LIN {X 0,Y 354.923,Z 398.899,A -85,B 0,C 180,E1 -13512.581,E2 -13512.581} C_VEL
LIN {X 0,Y 354.894,Z 398.905,A -85,B 0,C 180,E1 -13516.096,E2 -13516.096} C_VEL
LIN {X 0,Y 354.908,Z 398.901,A -85,B 0,C 180,E1 -13518.472,E2 -13518.472} C_VEL
LIN {X 0,Y 354.836,Z 398.91,A -85,B 0,C 180,E1 -13522.106,E2 -13522.106} C_VEL
LIN {X 0,Y 354.9,Z 398.904,A -85,B 0,C 180,E1 -13525.827,E2 -13525.827} C_VEL
LIN {X 0,Y 354.819,Z 398.912,A -85,B 0,C 180,E1 -13529.682,E2 -13529.682} C_VEL
LIN {X 0,Y 354.807,Z 398.915,A -85,B 0,C 180,E1 -13533.702,E2 -13533.702} C_VEL
LIN {X 0,Y 354.803,Z 398.914,A -85,B 0,C 180,E1 -13536.459,E2 -13536.459} C_VEL
LIN {X 0,Y 354.825,Z 398.912,A -85,B 0,C 180,E1 -13539.424,E2 -13539.424} C_VEL
LIN {X 0,Y 354.79,Z 398.917,A -85,B 0,C 180,E1 -13542.867,E2 -13542.867} C_VEL
LIN {X 0,Y 354.779,Z 398.919,A -85,B 0,C 180,E1 -13546.105,E2 -13546.105} C_VEL
LIN {X 0,Y 354.854,Z 399.148,A -85,B 0,C 180,E1 -13547.122,E2 -13547.122} C_VEL
LIN {X 0,Y 355.19,Z 402.697,A -85,B 0,C 180,E1 -13550.505,E2 -13550.505} C_VEL
LIN {X 0,Y 355.149,Z 406.159,A -85,B 0,C 180,E1 -13553.582,E2 -13553.582} C_VEL
LIN {X 0,Y 354.934,Z 409.364,A -85,B 0,C 180,E1 -13556.329,E2 -13556.329} C_VEL
LIN {X 0,Y 354.662,Z 412.578,A -85,B 0,C 180,E1 -13558.988,E2 -13558.988} C_VEL
LIN {X 0,Y 354.41,Z 415.78,A -85,B 0,C 180,E1 -13561.581,E2 -13561.581} C_VEL
LIN {X 0,Y 354.107,Z 420.28,A -85,B 0,C 180,E1 -13565.134,E2 -13565.134} C_VEL
LIN {X 0,Y 358.979,Z 436.572,A -85,B 0,C 180,E1 -13566.069,E2 -13566.069} C_VEL
LIN {X 0,Y 362.051,Z 449.481,A -85,B 0,C 180,E1 -13566.956,E2 -13566.956} C_VEL
LIN {X 0,Y 363.817,Z 459.076,A -85,B 0,C 180,E1 -13567.713,E2 -13567.713} C_VEL
LIN {X 0,Y 363.535,Z 464.599,A -85,B 0,C 180,E1 -13568.119,E2 -13568.119} C_VEL
LIN {X 0,Y 362.37,Z 476.477,A -85,B 0,C 180,E1 -13569.122,E2 -13569.122} C_VEL
LIN {X 0,Y 360.894,Z 488.433,A -85,B 0,C 180,E1 -13570.371,E2 -13570.371} C_VEL
LIN {X 0,Y 359.361,Z 499.34,A -85,B 0,C 180,E1 -13571.765,E2 -13571.765} C_VEL
LIN {X 0,Y 357.822,Z 510.101,A -85,B 0,C 180,E1 -13573.453,E2 -13573.453} C_VEL
LIN {X 0,Y 356.582,Z 518.981,A -85,B 0,C 180,E1 -13575.154,E2 -13575.154} C_VEL
LIN {X 0,Y 355.662,Z 526.369,A -85,B 0,C 180,E1 -13576.865,E2 -13576.865} C_VEL
LIN {X 0,Y 354.749,Z 532.527,A -85,B 0,C 180,E1 -13578.574,E2 -13578.574} C_VEL
LIN {X 0,Y 354.17,Z 537.615,A -85,B 0,C 180,E1 -13580.29,E2 -13580.29} C_VEL
LIN {X 0,Y 353.634,Z 542.891,A -85,B 0,C 180,E1 -13582.578,E2 -13582.578} C_VEL
LIN {X 0,Y 353.426,Z 545.835,A -85,B 0,C 180,E1 -13584.294,E2 -13584.294} C_VEL
LIN {X 0,Y 353.232,Z 548.54,A -85,B 0,C 180,E1 -13586.578,E2 -13586.578} C_VEL
LIN {X 0,Y 353.157,Z 549.895,A -85,B 0,C 180,E1 -13588.86,E2 -13588.86} C_VEL
LIN {X 0,Y 353.157,Z 549.928,A -85,B 0,C 180,E1 -13591.14,E2 -13591.14} C_VEL
LIN {X 0,Y 353.231,Z 548.635,A -85,B 0,C 180,E1 -13593.422,E2 -13593.422} C_VEL
LIN {X 0,Y 353.424,Z 545.987,A -85,B 0,C 180,E1 -13595.706,E2 -13595.706} C_VEL
LIN {X 0,Y 353.721,Z 541.916,A -85,B 0,C 180,E1 -13597.995,E2 -13597.995} C_VEL
LIN {X 0,Y 354.314,Z 536.291,A -85,B 0,C 180,E1 -13600.284,E2 -13600.284} C_VEL
LIN {X 0,Y 355.115,Z 529.94,A -85,B 0,C 180,E1 -13602.284,E2 -13602.284} C_VEL
LIN {X 0,Y 356.245,Z 522.042,A -85,B 0,C 180,E1 -13604.277,E2 -13604.277} C_VEL
LIN {X 0,Y 357.339,Z 513.781,A -85,B 0,C 180,E1 -13605.983,E2 -13605.983} C_VEL
LIN {X 0,Y 358.781,Z 503.825,A -85,B 0,C 180,E1 -13607.675,E2 -13607.675} C_VEL
LIN {X 0,Y 360.336,Z 492.742,A -85,B 0,C 180,E1 -13609.216,E2 -13609.216} C_VEL
LIN {X 0,Y 361.75,Z 481.707,A -85,B 0,C 180,E1 -13610.469,E2 -13610.469} C_VEL
LIN {X 0,Y 363.134,Z 469.725,A -85,B 0,C 180,E1 -13611.575,E2 -13611.575} C_VEL
LIN {X 0,Y 363.949,Z 460.574,A -85,B 0,C 180,E1 -13612.269,E2 -13612.269} C_VEL
LIN {X 0,Y 362.131,Z 449.749,A -85,B 0,C 180,E1 -13613.128,E2 -13613.128} C_VEL
LIN {X 0,Y 358.864,Z 436.14,A -85,B 0,C 180,E1 -13614.063,E2 -13614.063} C_VEL
LIN {X 0,Y 354.669,Z 422.615,A -85,B 0,C 180,E1 -13614.849,E2 -13614.849} C_VEL
LIN {X 0,Y 354.099,Z 420.265,A -85,B 0,C 180,E1 -13614.985,E2 -13614.985} C_VEL
LIN {X 0,Y 354.31,Z 417.51,A -85,B 0,C 180,E1 -13617.144,E2 -13617.144} C_VEL
LIN {X 0,Y 354.66,Z 412.711,A -85,B 0,C 180,E1 -13621.012,E2 -13621.012} C_VEL
LIN {X 0,Y 354.928,Z 409.411,A -85,B 0,C 180,E1 -13623.731,E2 -13623.731} C_VEL
LIN {X 0,Y 355.142,Z 405.684,A -85,B 0,C 180,E1 -13626.92,E2 -13626.92} C_VEL
LIN {X 0,Y 354.513,Z 404.734,A -85,B 0,C 180,E1 -13627.855,E2 -13627.855} C_VEL
LIN {X 0,Y 351.722,Z 403.491,A -85,B 0,C 180,E1 -13629.385,E2 -13629.385} C_VEL
LIN {X 0,Y 349.277,Z 402.535,A -85,B 0,C 180,E1 -13630.623,E2 -13630.623} C_VEL
LIN {X 0,Y 348.133,Z 401.704,A -85,B 0,C 180,E1 -13631.578,E2 -13631.578} C_VEL
LIN {X 0,Y 347.99,Z 401.39,A -85,B 0,C 180,E1 -13631.901,E2 -13631.901} C_VEL
LIN {X 0,Y 347.786,Z 399.889,A -85,B 0,C 180,E1 -13633.399,E2 -13633.399} C_VEL
LIN {X 0,Y 347.728,Z 399.801,A -85,B 0,C 180,E1 -13636.686,E2 -13636.686} C_VEL
LIN {X 0,Y 347.749,Z 399.794,A -85,B 0,C 180,E1 -13640.173,E2 -13640.173} C_VEL
LIN {X 0,Y 347.765,Z 399.793,A -85,B 0,C 180,E1 -13642.679,E2 -13642.679} C_VEL
LIN {X 0,Y 347.75,Z 399.793,A -85,B 0,C 180,E1 -13645.956,E2 -13645.956} C_VEL
LIN {X 0,Y 347.766,Z 399.791,A -85,B 0,C 180,E1 -13649.654,E2 -13649.654} C_VEL
LIN {X 0,Y 347.853,Z 399.782,A -85,B 0,C 180,E1 -13652.745,E2 -13652.745} C_VEL
LIN {X 0,Y 347.791,Z 399.785,A -85,B 0,C 180,E1 -13656.162,E2 -13656.162} C_VEL
LIN {X 0,Y 347.82,Z 399.779,A -85,B 0,C 180,E1 -13659.91,E2 -13659.91} C_VEL
LIN {X 0,Y 347.869,Z 399.779,A -85,B 0,C 180,E1 -13662.359,E2 -13662.359} C_VEL
LIN {X 0,Y 347.9,Z 399.773,A -85,B 0,C 180,E1 -13665.971,E2 -13665.971} C_VEL
LIN {X 0,Y 347.931,Z 399.769,A -85,B 0,C 180,E1 -13669.526,E2 -13669.526} C_VEL
LIN {X 0,Y 348.077,Z 399.753,A -85,B 0,C 180,E1 -13671.875,E2 -13671.875} C_VEL
LIN {X 0,Y 348.07,Z 399.752,A -85,B 0,C 180,E1 -13674.206,E2 -13674.206} C_VEL
LIN {X 0,Y 348.209,Z 399.735,A -85,B 0,C 180,E1 -13677.686,E2 -13677.686} C_VEL
LIN {X 0,Y 348.348,Z 399.721,A -85,B 0,C 180,E1 -13680,E2 -13680} C_VEL
LIN {X 0,Y 348.211,Z 399.735,A -85,B 0,C 180,E1 -13682.313,E2 -13682.313} C_VEL
LIN {X 0,Y 348.109,Z 399.748,A -85,B 0,C 180,E1 -13686.957,E2 -13686.957} C_VEL
LIN {X 0,Y 347.971,Z 399.766,A -85,B 0,C 180,E1 -13689.298,E2 -13689.298} C_VEL
LIN {X 0,Y 347.893,Z 399.776,A -85,B 0,C 180,E1 -13692.839,E2 -13692.839} C_VEL
LIN {X 0,Y 347.842,Z 399.782,A -85,B 0,C 180,E1 -13696.431,E2 -13696.431} C_VEL
LIN {X 0,Y 347.858,Z 399.779,A -85,B 0,C 180,E1 -13698.86,E2 -13698.86} C_VEL
LIN {X 0,Y 347.776,Z 399.791,A -85,B 0,C 180,E1 -13702.579,E2 -13702.579} C_VEL
LIN {X 0,Y 347.814,Z 399.784,A -85,B 0,C 180,E1 -13705.108,E2 -13705.108} C_VEL
LIN {X 0,Y 347.81,Z 399.784,A -85,B 0,C 180,E1 -13707.694,E2 -13707.694} C_VEL
LIN {X 0,Y 347.751,Z 399.79,A -85,B 0,C 180,E1 -13710.348,E2 -13710.348} C_VEL
LIN {X 0,Y 347.75,Z 399.796,A -85,B 0,C 180,E1 -13714.044,E2 -13714.044} C_VEL
LIN {X 0,Y 347.769,Z 399.796,A -85,B 0,C 180,E1 -13717.32,E2 -13717.32} C_VEL
LIN {X 0,Y 347.757,Z 399.797,A -85,B 0,C 180,E1 -13720.294,E2 -13720.294} C_VEL
LIN {X 0,Y 347.785,Z 399.804,A -85,B 0,C 180,E1 -13723.999,E2 -13723.999} C_VEL
LIN {X 0,Y 348.233,Z 402.702,A -85,B 0,C 180,E1 -13726.671,E2 -13726.671} C_VEL
LIN {X 0,Y 348.67,Z 406.35,A -85,B 0,C 180,E1 -13729.833,E2 -13729.833} C_VEL
LIN {X 0,Y 348.579,Z 409.986,A -85,B 0,C 180,E1 -13732.781,E2 -13732.781} C_VEL
LIN {X 0,Y 348.24,Z 413.96,A -85,B 0,C 180,E1 -13735.837,E2 -13735.837} C_VEL
LIN {X 0,Y 347.717,Z 419.139,A -85,B 0,C 180,E1 -13739.649,E2 -13739.649} C_VEL
LIN {X 0,Y 347.25,Z 424.619,A -85,B 0,C 180,E1 -13743.56,E2 -13743.56} C_VEL
LIN {X 0,Y 347.141,Z 426.014,A -85,B 0,C 180,E1 -13744.533,E2 -13744.533} C_VEL
LIN {X 0,Y 351.781,Z 442.131,A -85,B 0,C 180,E1 -13745.454,E2 -13745.454} C_VEL
LIN {X 0,Y 354.766,Z 455.294,A -85,B 0,C 180,E1 -13746.359,E2 -13746.359} C_VEL
LIN {X 0,Y 356.927,Z 468.457,A -85,B 0,C 180,E1 -13747.423,E2 -13747.423} C_VEL
LIN {X 0,Y 355.707,Z 481.093,A -85,B 0,C 180,E1 -13748.465,E2 -13748.465} C_VEL
LIN {X 0,Y 354.168,Z 492.999,A -85,B 0,C 180,E1 -13749.68,E2 -13749.68} C_VEL
LIN {X 0,Y 352.564,Z 504.301,A -85,B 0,C 180,E1 -13751.099,E2 -13751.099} C_VEL
LIN {X 0,Y 350.942,Z 515.371,A -85,B 0,C 180,E1 -13752.819,E2 -13752.819} C_VEL
LIN {X 0,Y 349.61,Z 524.504,A -85,B 0,C 180,E1 -13754.552,E2 -13754.552} C_VEL
LIN {X 0,Y 348.47,Z 533.233,A -85,B 0,C 180,E1 -13756.589,E2 -13756.589} C_VEL
LIN {X 0,Y 347.515,Z 539.378,A -85,B 0,C 180,E1 -13758.332,E2 -13758.332} C_VEL
LIN {X 0,Y 346.806,Z 545.907,A -85,B 0,C 180,E1 -13760.67,E2 -13760.67} C_VEL
LIN {X 0,Y 346.342,Z 550.793,A -85,B 0,C 180,E1 -13763.007,E2 -13763.007} C_VEL
LIN {X 0,Y 346.157,Z 554.19,A -85,B 0,C 180,E1 -13765.342,E2 -13765.342} C_VEL
LIN {X 0,Y 346.045,Z 556.198,A -85,B 0,C 180,E1 -13767.672,E2 -13767.672} C_VEL
LIN {X 0,Y 346.074,Z 556.862,A -85,B 0,C 180,E1 -13770,E2 -13770} C_VEL
LIN {X 0,Y 346.045,Z 556.192,A -85,B 0,C 180,E1 -13772.328,E2 -13772.328} C_VEL
LIN {X 0,Y 346.16,Z 554.18,A -85,B 0,C 180,E1 -13774.658,E2 -13774.658} C_VEL
LIN {X 0,Y 346.371,Z 550.776,A -85,B 0,C 180,E1 -13776.993,E2 -13776.993} C_VEL
LIN {X 0,Y 346.786,Z 545.877,A -85,B 0,C 180,E1 -13779.33,E2 -13779.33} C_VEL
LIN {X 0,Y 347.315,Z 541.154,A -85,B 0,C 180,E1 -13781.083,E2 -13781.083} C_VEL
LIN {X 0,Y 348.309,Z 534.306,A -85,B 0,C 180,E1 -13783.12,E2 -13783.12} C_VEL
LIN {X 0,Y 349.38,Z 525.802,A -85,B 0,C 180,E1 -13785.159,E2 -13785.159} C_VEL
LIN {X 0,Y 350.687,Z 516.931,A -85,B 0,C 180,E1 -13786.893,E2 -13786.893} C_VEL
LIN {X 0,Y 352.278,Z 506.184,A -85,B 0,C 180,E1 -13788.615,E2 -13788.615} C_VEL
LIN {X 0,Y 353.858,Z 495.308,A -85,B 0,C 180,E1 -13790.036,E2 -13790.036} C_VEL
LIN {X 0,Y 355.434,Z 483.058,A -85,B 0,C 180,E1 -13791.341,E2 -13791.341} C_VEL
LIN {X 0,Y 356.807,Z 470.278,A -85,B 0,C 180,E1 -13792.429,E2 -13792.429} C_VEL
LIN {X 0,Y 356.602,Z 466.361,A -85,B 0,C 180,E1 -13792.745,E2 -13792.745} C_VEL
LIN {X 0,Y 354.228,Z 452.721,A -85,B 0,C 180,E1 -13793.816,E2 -13793.816} C_VEL
LIN {X 0,Y 351.015,Z 439.421,A -85,B 0,C 180,E1 -13794.703,E2 -13794.703} C_VEL
LIN {X 0,Y 347.23,Z 426.891,A -85,B 0,C 180,E1 -13795.406,E2 -13795.406} C_VEL
LIN {X 0,Y 347.125,Z 426.008,A -85,B 0,C 180,E1 -13795.456,E2 -13795.456} C_VEL
LIN {X 0,Y 347.564,Z 420.929,A -85,B 0,C 180,E1 -13799.032,E2 -13799.032} C_VEL
LIN {X 0,Y 348.081,Z 415.449,A -85,B 0,C 180,E1 -13803.035,E2 -13803.035} C_VEL
LIN {X 0,Y 348.502,Z 411.233,A -85,B 0,C 180,E1 -13806.23,E2 -13806.23} C_VEL
LIN {X 0,Y 348.675,Z 408.132,A -85,B 0,C 180,E1 -13808.671,E2 -13808.671} C_VEL
LIN {X 0,Y 348.668,Z 406.318,A -85,B 0,C 180,E1 -13810.167,E2 -13810.167} C_VEL
LIN {X 0,Y 348.201,Z 402.67,A -85,B 0,C 180,E1 -13813.334,E2 -13813.334} C_VEL
LIN {X 0,Y 347.784,Z 399.794,A -85,B 0,C 180,E1 -13816.001,E2 -13816.001} C_VEL
LIN {X 0,Y 347.756,Z 399.795,A -85,B 0,C 180,E1 -13819.706,E2 -13819.706} C_VEL
LIN {X 0,Y 347.768,Z 399.794,A -85,B 0,C 180,E1 -13822.68,E2 -13822.68} C_VEL
LIN {X 0,Y 347.749,Z 399.796,A -85,B 0,C 180,E1 -13825.956,E2 -13825.956} C_VEL
LIN {X 0,Y 347.75,Z 399.795,A -85,B 0,C 180,E1 -13829.652,E2 -13829.652} C_VEL
LIN {X 0,Y 347.831,Z 399.784,A -85,B 0,C 180,E1 -13833.608,E2 -13833.608} C_VEL
LIN {X 0,Y 347.786,Z 399.789,A -85,B 0,C 180,E1 -13836.162,E2 -13836.162} C_VEL
LIN {X 0,Y 347.813,Z 399.784,A -85,B 0,C 180,E1 -13839.909,E2 -13839.909} C_VEL
LIN {X 0,Y 347.868,Z 399.777,A -85,B 0,C 180,E1 -13842.359,E2 -13842.359} C_VEL
LIN {X 0,Y 347.898,Z 399.773,A -85,B 0,C 180,E1 -13845.971,E2 -13845.971} C_VEL
LIN {X 0,Y 347.93,Z 399.767,A -85,B 0,C 180,E1 -13849.526,E2 -13849.526} C_VEL
LIN {X 0,Y 348.076,Z 399.751,A -85,B 0,C 180,E1 -13851.875,E2 -13851.875} C_VEL
LIN {X 0,Y 348.069,Z 399.752,A -85,B 0,C 180,E1 -13854.206,E2 -13854.206} C_VEL
LIN {X 0,Y 348.21,Z 399.734,A -85,B 0,C 180,E1 -13857.687,E2 -13857.687} C_VEL
LIN {X 0,Y 348.369,Z 399.717,A -85,B 0,C 180,E1 -13860,E2 -13860} C_VEL
LIN {X 0,Y 348.208,Z 399.734,A -85,B 0,C 180,E1 -13862.314,E2 -13862.314} C_VEL
LIN {X 0,Y 348.108,Z 399.748,A -85,B 0,C 180,E1 -13866.958,E2 -13866.958} C_VEL
LIN {X 0,Y 347.97,Z 399.765,A -85,B 0,C 180,E1 -13869.299,E2 -13869.299} C_VEL
LIN {X 0,Y 347.892,Z 399.774,A -85,B 0,C 180,E1 -13872.84,E2 -13872.84} C_VEL
LIN {X 0,Y 347.843,Z 399.779,A -85,B 0,C 180,E1 -13876.431,E2 -13876.431} C_VEL
LIN {X 0,Y 347.857,Z 399.779,A -85,B 0,C 180,E1 -13878.86,E2 -13878.86} C_VEL
LIN {X 0,Y 347.776,Z 399.792,A -85,B 0,C 180,E1 -13882.579,E2 -13882.579} C_VEL
LIN {X 0,Y 347.813,Z 399.784,A -85,B 0,C 180,E1 -13885.108,E2 -13885.108} C_VEL
LIN {X 0,Y 347.809,Z 399.788,A -85,B 0,C 180,E1 -13887.694,E2 -13887.694} C_VEL
LIN {X 0,Y 347.75,Z 399.792,A -85,B 0,C 180,E1 -13890.348,E2 -13890.348} C_VEL
LIN {X 0,Y 347.749,Z 399.795,A -85,B 0,C 180,E1 -13894.044,E2 -13894.044} C_VEL
LIN {X 0,Y 347.767,Z 399.793,A -85,B 0,C 180,E1 -13897.32,E2 -13897.32} C_VEL
LIN {X 0,Y 347.734,Z 399.796,A -85,B 0,C 180,E1 -13900.297,E2 -13900.297} C_VEL
LIN {X 0,Y 347.727,Z 399.797,A -85,B 0,C 180,E1 -13903.408,E2 -13903.408} C_VEL
LIN {X 0,Y 347.778,Z 399.85,A -85,B 0,C 180,E1 -13906.677,E2 -13906.677} C_VEL
LIN {X 0,Y 348.152,Z 403.345,A -85,B 0,C 180,E1 -13910.094,E2 -13910.094} C_VEL
LIN {X 0,Y 348.127,Z 406.196,A -85,B 0,C 180,E1 -13912.725,E2 -13912.725} C_VEL
LIN {X 0,Y 347.921,Z 409.844,A -85,B 0,C 180,E1 -13915.915,E2 -13915.915} C_VEL
LIN {X 0,Y 347.545,Z 414.23,A -85,B 0,C 180,E1 -13919.632,E2 -13919.632} C_VEL
LIN {X 0,Y 347.205,Z 419.05,A -85,B 0,C 180,E1 -13923.557,E2 -13923.557} C_VEL
LIN {X 0,Y 347.099,Z 420.355,A -85,B 0,C 180,E1 -13924.602,E2 -13924.602} C_VEL
LIN {X 0,Y 352.04,Z 436.533,A -85,B 0,C 180,E1 -13925.561,E2 -13925.561} C_VEL
LIN {X 0,Y 355.127,Z 449.404,A -85,B 0,C 180,E1 -13926.47,E2 -13926.47} C_VEL
LIN {X 0,Y 357.249,Z 461.563,A -85,B 0,C 180,E1 -13927.466,E2 -13927.466} C_VEL
LIN {X 0,Y 355.922,Z 475.051,A -85,B 0,C 180,E1 -13928.574,E2 -13928.574} C_VEL
LIN {X 0,Y 354.375,Z 487.327,A -85,B 0,C 180,E1 -13929.844,E2 -13929.844} C_VEL
LIN {X 0,Y 352.844,Z 497.419,A -85,B 0,C 180,E1 -13931.115,E2 -13931.115} C_VEL
LIN {X 0,Y 351.507,Z 506.838,A -85,B 0,C 180,E1 -13932.548,E2 -13932.548} C_VEL
LIN {X 0,Y 350.09,Z 516.305,A -85,B 0,C 180,E1 -13934.276,E2 -13934.276} C_VEL
LIN {X 0,Y 348.91,Z 525.327,A -85,B 0,C 180,E1 -13936.31,E2 -13936.31} C_VEL
LIN {X 0,Y 347.752,Z 532.598,A -85,B 0,C 180,E1 -13938.34,E2 -13938.34} C_VEL
LIN {X 0,Y 347.135,Z 537.686,A -85,B 0,C 180,E1 -13940.091,E2 -13940.091} C_VEL
LIN {X 0,Y 346.56,Z 542.961,A -85,B 0,C 180,E1 -13942.426,E2 -13942.426} C_VEL
LIN {X 0,Y 346.345,Z 545.904,A -85,B 0,C 180,E1 -13944.177,E2 -13944.177} C_VEL
LIN {X 0,Y 346.159,Z 548.609,A -85,B 0,C 180,E1 -13946.508,E2 -13946.508} C_VEL
LIN {X 0,Y 346.06,Z 549.964,A -85,B 0,C 180,E1 -13948.836,E2 -13948.836} C_VEL
LIN {X 0,Y 346.06,Z 549.997,A -85,B 0,C 180,E1 -13951.164,E2 -13951.164} C_VEL
LIN {X 0,Y 346.158,Z 548.704,A -85,B 0,C 180,E1 -13953.492,E2 -13953.492} C_VEL
LIN {X 0,Y 346.341,Z 546.055,A -85,B 0,C 180,E1 -13955.823,E2 -13955.823} C_VEL
LIN {X 0,Y 346.663,Z 541.984,A -85,B 0,C 180,E1 -13958.159,E2 -13958.159} C_VEL
LIN {X 0,Y 347.303,Z 536.359,A -85,B 0,C 180,E1 -13960.494,E2 -13960.494} C_VEL
LIN {X 0,Y 348.178,Z 530.007,A -85,B 0,C 180,E1 -13962.532,E2 -13962.532} C_VEL
LIN {X 0,Y 349.2,Z 523.337,A -85,B 0,C 180,E1 -13964.273,E2 -13964.273} C_VEL
LIN {X 0,Y 350.255,Z 515.478,A -85,B 0,C 180,E1 -13965.986,E2 -13965.986} C_VEL
LIN {X 0,Y 351.728,Z 505.67,A -85,B 0,C 180,E1 -13967.741,E2 -13967.741} C_VEL
LIN {X 0,Y 353.314,Z 494.948,A -85,B 0,C 180,E1 -13969.311,E2 -13969.311} C_VEL
LIN {X 0,Y 354.92,Z 483.066,A -85,B 0,C 180,E1 -13970.73,E2 -13970.73} C_VEL
LIN {X 0,Y 356.347,Z 471.396,A -85,B 0,C 180,E1 -13971.854,E2 -13971.854} C_VEL
LIN {X 0,Y 357.243,Z 460.637,A -85,B 0,C 180,E1 -13972.711,E2 -13972.711} C_VEL
LIN {X 0,Y 354.86,Z 448.199,A -85,B 0,C 180,E1 -13973.726,E2 -13973.726} C_VEL
LIN {X 0,Y 351.56,Z 434.852,A -85,B 0,C 180,E1 -13974.654,E2 -13974.654} C_VEL
LIN {X 0,Y 347.095,Z 420.357,A -85,B 0,C 180,E1 -13975.505,E2 -13975.505} C_VEL
LIN {X 0,Y 347.407,Z 415.979,A -85,B 0,C 180,E1 -13979.047,E2 -13979.047} C_VEL
LIN {X 0,Y 347.695,Z 412.513,A -85,B 0,C 180,E1 -13981.902,E2 -13981.902} C_VEL
LIN {X 0,Y 347.925,Z 409.517,A -85,B 0,C 180,E1 -13984.444,E2 -13984.444} C_VEL
LIN {X 0,Y 348.129,Z 406.326,A -85,B 0,C 180,E1 -13987.275,E2 -13987.275} C_VEL
LIN {X 0,Y 348.144,Z 403.115,A -85,B 0,C 180,E1 -13990.24,E2 -13990.24} C_VEL
LIN {X 0,Y 347.99,Z 401.39,A -85,B 0,C 180,E1 -13991.901,E2 -13991.901} C_VEL
LIN {X 0,Y 347.159,Z 400.689,A -85,B 0,C 180,E1 -13992.857,E2 -13992.857} C_VEL
LIN {X 0,Y 344.17,Z 400.394,A -85,B 0,C 180,E1 -13994.423,E2 -13994.423} C_VEL
LIN {X 0,Y 341.743,Z 400.551,A -85,B 0,C 180,E1 -13995.697,E2 -13995.697} C_VEL
LIN {X 0,Y 340.74,Z 400.672,A -85,B 0,C 180,E1 -13996.683,E2 -13996.683} C_VEL
LIN {X 0,Y 340.674,Z 400.679,A -85,B 0,C 180,E1 -13997.017,E2 -13997.017} C_VEL
LIN {X 0,Y 340.701,Z 400.672,A -85,B 0,C 180,E1 -14000.248,E2 -14000.248} C_VEL
LIN {X 0,Y 340.713,Z 400.669,A -85,B 0,C 180,E1 -14003.559,E2 -14003.559} C_VEL
LIN {X 0,Y 340.696,Z 400.673,A -85,B 0,C 180,E1 -14006.154,E2 -14006.154} C_VEL
LIN {X 0,Y 340.777,Z 400.661,A -85,B 0,C 180,E1 -14010.333,E2 -14010.333} C_VEL
LIN {X 0,Y 340.806,Z 400.658,A -85,B 0,C 180,E1 -14013.02,E2 -14013.02} C_VEL
LIN {X 0,Y 340.731,Z 400.665,A -85,B 0,C 180,E1 -14016.927,E2 -14016.927} C_VEL
LIN {X 0,Y 340.797,Z 400.66,A -85,B 0,C 180,E1 -14020.734,E2 -14020.734} C_VEL
LIN {X 0,Y 340.789,Z 400.659,A -85,B 0,C 180,E1 -14023.219,E2 -14023.219} C_VEL
LIN {X 0,Y 340.847,Z 400.653,A -85,B 0,C 180,E1 -14026.89,E2 -14026.89} C_VEL
LIN {X 0,Y 340.931,Z 400.642,A -85,B 0,C 180,E1 -14030.508,E2 -14030.508} C_VEL
LIN {X 0,Y 341.079,Z 400.623,A -85,B 0,C 180,E1 -14032.898,E2 -14032.898} C_VEL
LIN {X 0,Y 341.171,Z 400.612,A -85,B 0,C 180,E1 -14037.639,E2 -14037.639} C_VEL
LIN {X 0,Y 341.298,Z 400.599,A -85,B 0,C 180,E1 -14040,E2 -14040} C_VEL
LIN {X 0,Y 341.173,Z 400.612,A -85,B 0,C 180,E1 -14042.361,E2 -14042.361} C_VEL
LIN {X 0,Y 341.079,Z 400.623,A -85,B 0,C 180,E1 -14047.102,E2 -14047.102} C_VEL
LIN {X 0,Y 340.875,Z 400.648,A -85,B 0,C 180,E1 -14050.694,E2 -14050.694} C_VEL
LIN {X 0,Y 340.865,Z 400.652,A -85,B 0,C 180,E1 -14054.325,E2 -14054.325} C_VEL
LIN {X 0,Y 340.84,Z 400.653,A -85,B 0,C 180,E1 -14058.467,E2 -14058.467} C_VEL
LIN {X 0,Y 340.756,Z 400.664,A -85,B 0,C 180,E1 -14061.857,E2 -14061.857} C_VEL
LIN {X 0,Y 340.774,Z 400.662,A -85,B 0,C 180,E1 -14065.664,E2 -14065.664} C_VEL
LIN {X 0,Y 340.73,Z 400.667,A -85,B 0,C 180,E1 -14068.321,E2 -14068.321} C_VEL
LIN {X 0,Y 340.7,Z 400.673,A -85,B 0,C 180,E1 -14071.044,E2 -14071.044} C_VEL
LIN {X 0,Y 340.721,Z 400.671,A -85,B 0,C 180,E1 -14075.279,E2 -14075.279} C_VEL
LIN {X 0,Y 340.722,Z 400.673,A -85,B 0,C 180,E1 -14078.388,E2 -14078.388} C_VEL
LIN {X 0,Y 340.735,Z 400.671,A -85,B 0,C 180,E1 -14082.052,E2 -14082.052} C_VEL
LIN {X 0,Y 340.757,Z 400.84,A -85,B 0,C 180,E1 -14083.791,E2 -14083.791} C_VEL
LIN {X 0,Y 341.295,Z 404.475,A -85,B 0,C 180,E1 -14087.192,E2 -14087.192} C_VEL
LIN {X 0,Y 341.657,Z 408.115,A -85,B 0,C 180,E1 -14090.381,E2 -14090.381} C_VEL
LIN {X 0,Y 341.514,Z 411.77,A -85,B 0,C 180,E1 -14093.377,E2 -14093.377} C_VEL
LIN {X 0,Y 341.131,Z 415.42,A -85,B 0,C 180,E1 -14096.202,E2 -14096.202} C_VEL
LIN {X 0,Y 340.615,Z 420.564,A -85,B 0,C 180,E1 -14100.066,E2 -14100.066} C_VEL
LIN {X 0,Y 340.134,Z 425.958,A -85,B 0,C 180,E1 -14103.983,E2 -14103.983} C_VEL
LIN {X 0,Y 341.878,Z 431.912,A -85,B 0,C 180,E1 -14104.295,E2 -14104.295} C_VEL
LIN {X 0,Y 345.815,Z 445.867,A -85,B 0,C 180,E1 -14105.18,E2 -14105.18} C_VEL
LIN {X 0,Y 348.571,Z 458.794,A -85,B 0,C 180,E1 -14106.14,E2 -14106.14} C_VEL
LIN {X 0,Y 350.244,Z 470.619,A -85,B 0,C 180,E1 -14107.147,E2 -14107.147} C_VEL
LIN {X 0,Y 348.795,Z 483.48,A -85,B 0,C 180,E1 -14108.271,E2 -14108.271} C_VEL
LIN {X 0,Y 347.136,Z 495.346,A -85,B 0,C 180,E1 -14109.559,E2 -14109.559} C_VEL
LIN {X 0,Y 345.518,Z 506.203,A -85,B 0,C 180,E1 -14111.007,E2 -14111.007} C_VEL
LIN {X 0,Y 343.862,Z 516.933,A -85,B 0,C 180,E1 -14112.761,E2 -14112.761} C_VEL
LIN {X 0,Y 342.511,Z 525.792,A -85,B 0,C 180,E1 -14114.529,E2 -14114.529} C_VEL
LIN {X 0,Y 341.517,Z 533.165,A -85,B 0,C 180,E1 -14116.311,E2 -14116.311} C_VEL
LIN {X 0,Y 340.537,Z 539.31,A -85,B 0,C 180,E1 -14118.09,E2 -14118.09} C_VEL
LIN {X 0,Y 339.764,Z 545.839,A -85,B 0,C 180,E1 -14120.475,E2 -14120.475} C_VEL
LIN {X 0,Y 339.272,Z 550.725,A -85,B 0,C 180,E1 -14122.86,E2 -14122.86} C_VEL
LIN {X 0,Y 339.064,Z 554.121,A -85,B 0,C 180,E1 -14125.244,E2 -14125.244} C_VEL
LIN {X 0,Y 338.961,Z 556.129,A -85,B 0,C 180,E1 -14127.623,E2 -14127.623} C_VEL
LIN {X 0,Y 338.977,Z 556.793,A -85,B 0,C 180,E1 -14130,E2 -14130} C_VEL
LIN {X 0,Y 338.961,Z 556.123,A -85,B 0,C 180,E1 -14132.377,E2 -14132.377} C_VEL
LIN {X 0,Y 339.066,Z 554.11,A -85,B 0,C 180,E1 -14134.756,E2 -14134.756} C_VEL
LIN {X 0,Y 339.29,Z 550.706,A -85,B 0,C 180,E1 -14137.139,E2 -14137.139} C_VEL
LIN {X 0,Y 339.749,Z 545.807,A -85,B 0,C 180,E1 -14139.525,E2 -14139.525} C_VEL
LIN {X 0,Y 340.535,Z 539.27,A -85,B 0,C 180,E1 -14141.91,E2 -14141.91} C_VEL
LIN {X 0,Y 341.625,Z 531.998,A -85,B 0,C 180,E1 -14143.988,E2 -14143.988} C_VEL
LIN {X 0,Y 342.945,Z 522.989,A -85,B 0,C 180,E1 -14146.061,E2 -14146.061} C_VEL
LIN {X 0,Y 344.417,Z 513.536,A -85,B 0,C 180,E1 -14147.823,E2 -14147.823} C_VEL
LIN {X 0,Y 346.016,Z 503.07,A -85,B 0,C 180,E1 -14149.426,E2 -14149.426} C_VEL
LIN {X 0,Y 347.704,Z 491.52,A -85,B 0,C 180,E1 -14150.87,E2 -14150.87} C_VEL
LIN {X 0,Y 349.273,Z 478.889,A -85,B 0,C 180,E1 -14152.147,E2 -14152.147} C_VEL
LIN {X 0,Y 350.172,Z 470.5,A -85,B 0,C 180,E1 -14152.853,E2 -14152.853} C_VEL
LIN {X 0,Y 348.423,Z 458.217,A -85,B 0,C 180,E1 -14153.894,E2 -14153.894} C_VEL
LIN {X 0,Y 345.412,Z 444.356,A -85,B 0,C 180,E1 -14154.911,E2 -14154.911} C_VEL
LIN {X 0,Y 341.509,Z 430.874,A -85,B 0,C 180,E1 -14155.752,E2 -14155.752} C_VEL
LIN {X 0,Y 340.117,Z 425.934,A -85,B 0,C 180,E1 -14156.018,E2 -14156.018} C_VEL
LIN {X 0,Y 340.596,Z 420.876,A -85,B 0,C 180,E1 -14159.685,E2 -14159.685} C_VEL
LIN {X 0,Y 340.944,Z 417.206,A -85,B 0,C 180,E1 -14162.408,E2 -14162.408} C_VEL
LIN {X 0,Y 341.315,Z 413.555,A -85,B 0,C 180,E1 -14165.208,E2 -14165.208} C_VEL
LIN {X 0,Y 341.601,Z 409.906,A -85,B 0,C 180,E1 -14168.113,E2 -14168.113} C_VEL
LIN {X 0,Y 341.613,Z 407.142,A -85,B 0,C 180,E1 -14170.43,E2 -14170.43} C_VEL
LIN {X 0,Y 341.129,Z 403.297,A -85,B 0,C 180,E1 -14173.857,E2 -14173.857} C_VEL
LIN {X 0,Y 340.741,Z 400.671,A -85,B 0,C 180,E1 -14176.434,E2 -14176.434} C_VEL
LIN {X 0,Y 340.711,Z 400.672,A -85,B 0,C 180,E1 -14180.249,E2 -14180.249} C_VEL
LIN {X 0,Y 340.713,Z 400.671,A -85,B 0,C 180,E1 -14183.559,E2 -14183.559} C_VEL
LIN {X 0,Y 340.695,Z 400.675,A -85,B 0,C 180,E1 -14186.154,E2 -14186.154} C_VEL
LIN {X 0,Y 340.742,Z 400.668,A -85,B 0,C 180,E1 -14190.329,E2 -14190.329} C_VEL
LIN {X 0,Y 340.804,Z 400.659,A -85,B 0,C 180,E1 -14193.02,E2 -14193.02} C_VEL
LIN {X 0,Y 340.755,Z 400.666,A -85,B 0,C 180,E1 -14195.638,E2 -14195.638} C_VEL
LIN {X 0,Y 340.738,Z 400.666,A -85,B 0,C 180,E1 -14199.474,E2 -14199.474} C_VEL
LIN {X 0,Y 340.86,Z 400.65,A -85,B 0,C 180,E1 -14201.984,E2 -14201.984} C_VEL
LIN {X 0,Y 340.87,Z 400.648,A -85,B 0,C 180,E1 -14205.705,E2 -14205.705} C_VEL
LIN {X 0,Y 340.872,Z 400.646,A -85,B 0,C 180,E1 -14209.306,E2 -14209.306} C_VEL
LIN {X 0,Y 341.077,Z 400.619,A -85,B 0,C 180,E1 -14212.898,E2 -14212.898} C_VEL
LIN {X 0,Y 341.172,Z 400.611,A -85,B 0,C 180,E1 -14217.639,E2 -14217.639} C_VEL
LIN {X 0,Y 341.318,Z 400.595,A -85,B 0,C 180,E1 -14220,E2 -14220} C_VEL
LIN {X 0,Y 341.169,Z 400.611,A -85,B 0,C 180,E1 -14222.361,E2 -14222.361} C_VEL
LIN {X 0,Y 341.077,Z 400.624,A -85,B 0,C 180,E1 -14227.102,E2 -14227.102} C_VEL
LIN {X 0,Y 340.874,Z 400.648,A -85,B 0,C 180,E1 -14230.694,E2 -14230.694} C_VEL
LIN {X 0,Y 340.864,Z 400.648,A -85,B 0,C 180,E1 -14234.325,E2 -14234.325} C_VEL
LIN {X 0,Y 340.839,Z 400.653,A -85,B 0,C 180,E1 -14238.467,E2 -14238.467} C_VEL
LIN {X 0,Y 340.755,Z 400.664,A -85,B 0,C 180,E1 -14241.857,E2 -14241.857} C_VEL
LIN {X 0,Y 340.774,Z 400.663,A -85,B 0,C 180,E1 -14245.664,E2 -14245.664} C_VEL
LIN {X 0,Y 340.729,Z 400.667,A -85,B 0,C 180,E1 -14248.321,E2 -14248.321} C_VEL
LIN {X 0,Y 340.699,Z 400.673,A -85,B 0,C 180,E1 -14251.045,E2 -14251.045} C_VEL
LIN {X 0,Y 340.72,Z 400.669,A -85,B 0,C 180,E1 -14255.279,E2 -14255.279} C_VEL
LIN {X 0,Y 340.713,Z 400.668,A -85,B 0,C 180,E1 -14258.387,E2 -14258.387} C_VEL
LIN {X 0,Y 340.7,Z 400.674,A -85,B 0,C 180,E1 -14262.046,E2 -14262.046} C_VEL
LIN {X 0,Y 340.693,Z 400.673,A -85,B 0,C 180,E1 -14265.463,E2 -14265.463} C_VEL
LIN {X 0,Y 340.69,Z 400.674,A -85,B 0,C 180,E1 -14266.221,E2 -14266.221} C_VEL
LIN {X 0,Y 341.121,Z 403.999,A -85,B 0,C 180,E1 -14269.668,E2 -14269.668} C_VEL
LIN {X 0,Y 341.124,Z 406.262,A -85,B 0,C 180,E1 -14271.824,E2 -14271.824} C_VEL
LIN {X 0,Y 340.975,Z 409.467,A -85,B 0,C 180,E1 -14274.752,E2 -14274.752} C_VEL
LIN {X 0,Y 340.683,Z 412.928,A -85,B 0,C 180,E1 -14277.758,E2 -14277.758} C_VEL
LIN {X 0,Y 340.319,Z 417.506,A -85,B 0,C 180,E1 -14281.642,E2 -14281.642} C_VEL
LIN {X 0,Y 340.093,Z 420.424,A -85,B 0,C 180,E1 -14284.034,E2 -14284.034} C_VEL
LIN {X 0,Y 345.183,Z 436.908,A -85,B 0,C 180,E1 -14285.055,E2 -14285.055} C_VEL
LIN {X 0,Y 348.492,Z 450.49,A -85,B 0,C 180,E1 -14286.056,E2 -14286.056} C_VEL
LIN {X 0,Y 350.533,Z 462.029,A -85,B 0,C 180,E1 -14287.04,E2 -14287.04} C_VEL
LIN {X 0,Y 349.297,Z 475.351,A -85,B 0,C 180,E1 -14288.169,E2 -14288.169} C_VEL
LIN {X 0,Y 347.701,Z 487.401,A -85,B 0,C 180,E1 -14289.44,E2 -14289.44} C_VEL
LIN {X 0,Y 346.109,Z 497.492,A -85,B 0,C 180,E1 -14290.733,E2 -14290.733} C_VEL
LIN {X 0,Y 344.735,Z 506.91,A -85,B 0,C 180,E1 -14292.194,E2 -14292.194} C_VEL
LIN {X 0,Y 343.223,Z 516.377,A -85,B 0,C 180,E1 -14293.953,E2 -14293.953} C_VEL
LIN {X 0,Y 341.994,Z 525.398,A -85,B 0,C 180,E1 -14296.027,E2 -14296.027} C_VEL
LIN {X 0,Y 340.761,Z 532.669,A -85,B 0,C 180,E1 -14298.098,E2 -14298.098} C_VEL
LIN {X 0,Y 340.115,Z 537.756,A -85,B 0,C 180,E1 -14299.884,E2 -14299.884} C_VEL
LIN {X 0,Y 339.509,Z 543.031,A -85,B 0,C 180,E1 -14302.267,E2 -14302.267} C_VEL
LIN {X 0,Y 339.279,Z 545.974,A -85,B 0,C 180,E1 -14304.055,E2 -14304.055} C_VEL
LIN {X 0,Y 339.087,Z 548.679,A -85,B 0,C 180,E1 -14306.435,E2 -14306.435} C_VEL
LIN {X 0,Y 338.966,Z 550.033,A -85,B 0,C 180,E1 -14308.812,E2 -14308.812} C_VEL
LIN {X 0,Y 338.966,Z 550.066,A -85,B 0,C 180,E1 -14311.188,E2 -14311.188} C_VEL
LIN {X 0,Y 339.086,Z 548.772,A -85,B 0,C 180,E1 -14313.565,E2 -14313.565} C_VEL
LIN {X 0,Y 339.279,Z 546.123,A -85,B 0,C 180,E1 -14315.945,E2 -14315.945} C_VEL
LIN {X 0,Y 339.608,Z 542.052,A -85,B 0,C 180,E1 -14318.329,E2 -14318.329} C_VEL
LIN {X 0,Y 340.306,Z 536.426,A -85,B 0,C 180,E1 -14320.712,E2 -14320.712} C_VEL
LIN {X 0,Y 341.242,Z 530.074,A -85,B 0,C 180,E1 -14322.791,E2 -14322.791} C_VEL
LIN {X 0,Y 342.372,Z 522.362,A -85,B 0,C 180,E1 -14324.822,E2 -14324.822} C_VEL
LIN {X 0,Y 343.657,Z 513.914,A -85,B 0,C 180,E1 -14326.637,E2 -14326.637} C_VEL
LIN {X 0,Y 345.201,Z 503.958,A -85,B 0,C 180,E1 -14328.395,E2 -14328.395} C_VEL
LIN {X 0,Y 346.928,Z 492.873,A -85,B 0,C 180,E1 -14329.99,E2 -14329.99} C_VEL
LIN {X 0,Y 348.662,Z 480.52,A -85,B 0,C 180,E1 -14331.419,E2 -14331.419} C_VEL
LIN {X 0,Y 350.165,Z 467.85,A -85,B 0,C 180,E1 -14332.594,E2 -14332.594} C_VEL
LIN {X 0,Y 350.492,Z 461.534,A -85,B 0,C 180,E1 -14333.108,E2 -14333.108} C_VEL
LIN {X 0,Y 348.191,Z 449.193,A -85,B 0,C 180,E1 -14334.153,E2 -14334.153} C_VEL
LIN {X 0,Y 344.978,Z 436.301,A -85,B 0,C 180,E1 -14335.095,E2 -14335.095} C_VEL
LIN {X 0,Y 340.744,Z 423.018,A -85,B 0,C 180,E1 -14335.93,E2 -14335.93} C_VEL
LIN {X 0,Y 340.104,Z 420.407,A -85,B 0,C 180,E1 -14336.089,E2 -14336.089} C_VEL
LIN {X 0,Y 340.409,Z 415.811,A -85,B 0,C 180,E1 -14339.874,E2 -14339.874} C_VEL
LIN {X 0,Y 340.69,Z 412.796,A -85,B 0,C 180,E1 -14342.436,E2 -14342.436} C_VEL
LIN {X 0,Y 340.967,Z 409.598,A -85,B 0,C 180,E1 -14345.25,E2 -14345.25} C_VEL
LIN {X 0,Y 341.133,Z 406.068,A -85,B 0,C 180,E1 -14348.475,E2 -14348.475} C_VEL
LIN {X 0,Y 341.05,Z 403.159,A -85,B 0,C 180,E1 -14351.256,E2 -14351.256} C_VEL
LIN {X 0,Y 340.708,Z 400.677,A -85,B 0,C 180,E1 -14353.783,E2 -14353.783} C_VEL
LIN {X 0,Y 340.674,Z 400.679,A -85,B 0,C 180,E1 -14357.017,E2 -14357.017} C_VEL
LIN {X 0,Y 340.038,Z 400.76,A -85,B 0,C 180,E1 -14358.003,E2 -14358.003} C_VEL
LIN {X 0,Y 337.17,Z 401.114,A -85,B 0,C 180,E1 -14359.606,E2 -14359.606} C_VEL
LIN {X 0,Y 334.737,Z 401.415,A -85,B 0,C 180,E1 -14360.905,E2 -14360.905} C_VEL
LIN {X 0,Y 333.717,Z 401.54,A -85,B 0,C 180,E1 -14361.911,E2 -14361.911} C_VEL
LIN {X 0,Y 333.65,Z 401.549,A -85,B 0,C 180,E1 -14362.251,E2 -14362.251} C_VEL
LIN {X 0,Y 333.676,Z 401.546,A -85,B 0,C 180,E1 -14365.341,E2 -14365.341} C_VEL
LIN {X 0,Y 333.705,Z 401.542,A -85,B 0,C 180,E1 -14369.71,E2 -14369.71} C_VEL
LIN {X 0,Y 333.745,Z 401.539,A -85,B 0,C 180,E1 -14372.401,E2 -14372.401} C_VEL
LIN {X 0,Y 333.729,Z 401.539,A -85,B 0,C 180,E1 -14375.091,E2 -14375.091} C_VEL
LIN {X 0,Y 333.689,Z 401.542,A -85,B 0,C 180,E1 -14379.02,E2 -14379.02} C_VEL
LIN {X 0,Y 333.797,Z 401.531,A -85,B 0,C 180,E1 -14381.59,E2 -14381.59} C_VEL
LIN {X 0,Y 333.811,Z 401.531,A -85,B 0,C 180,E1 -14385.576,E2 -14385.576} C_VEL
LIN {X 0,Y 333.837,Z 401.526,A -85,B 0,C 180,E1 -14389.078,E2 -14389.078} C_VEL
LIN {X 0,Y 334.028,Z 401.501,A -85,B 0,C 180,E1 -14392.747,E2 -14392.747} C_VEL
LIN {X 0,Y 333.813,Z 401.53,A -85,B 0,C 180,E1 -14395.169,E2 -14395.169} C_VEL
LIN {X 0,Y 334.108,Z 401.491,A -85,B 0,C 180,E1 -14397.589,E2 -14397.589} C_VEL
LIN {X 0,Y 334.249,Z 401.477,A -85,B 0,C 180,E1 -14400,E2 -14400} C_VEL
LIN {X 0,Y 334.11,Z 401.491,A -85,B 0,C 180,E1 -14402.411,E2 -14402.411} C_VEL
LIN {X 0,Y 334.028,Z 401.501,A -85,B 0,C 180,E1 -14407.252,E2 -14407.252} C_VEL
LIN {X 0,Y 333.837,Z 401.525,A -85,B 0,C 180,E1 -14410.922,E2 -14410.922} C_VEL
LIN {X 0,Y 333.811,Z 401.53,A -85,B 0,C 180,E1 -14414.634,E2 -14414.634} C_VEL
LIN {X 0,Y 333.799,Z 401.53,A -85,B 0,C 180,E1 -14418.655,E2 -14418.655} C_VEL
LIN {X 0,Y 333.694,Z 401.544,A -85,B 0,C 180,E1 -14422.278,E2 -14422.278} C_VEL
LIN {X 0,Y 333.737,Z 401.537,A -85,B 0,C 180,E1 -14426.246,E2 -14426.246} C_VEL
LIN {X 0,Y 333.692,Z 401.546,A -85,B 0,C 180,E1 -14428.974,E2 -14428.974} C_VEL
LIN {X 0,Y 333.647,Z 401.552,A -85,B 0,C 180,E1 -14432.587,E2 -14432.587} C_VEL
LIN {X 0,Y 333.679,Z 401.55,A -85,B 0,C 180,E1 -14436.139,E2 -14436.139} C_VEL
LIN {X 0,Y 333.675,Z 401.552,A -85,B 0,C 180,E1 -14439.188,E2 -14439.188} C_VEL
LIN {X 0,Y 333.733,Z 401.707,A -85,B 0,C 180,E1 -14443.409,E2 -14443.409} C_VEL
LIN {X 0,Y 334.146,Z 404.426,A -85,B 0,C 180,E1 -14446.046,E2 -14446.046} C_VEL
LIN {X 0,Y 334.575,Z 408.057,A -85,B 0,C 180,E1 -14449.369,E2 -14449.369} C_VEL
LIN {X 0,Y 334.636,Z 409.927,A -85,B 0,C 180,E1 -14450.993,E2 -14450.993} C_VEL
LIN {X 0,Y 334.387,Z 413.522,A -85,B 0,C 180,E1 -14453.95,E2 -14453.95} C_VEL
LIN {X 0,Y 333.929,Z 417.83,A -85,B 0,C 180,E1 -14457.336,E2 -14457.336} C_VEL
LIN {X 0,Y 333.429,Z 422.657,A -85,B 0,C 180,E1 -14461.001,E2 -14461.001} C_VEL
LIN {X 0,Y 333.17,Z 425.891,A -85,B 0,C 180,E1 -14463.392,E2 -14463.392} C_VEL
LIN {X 0,Y 334.892,Z 431.833,A -85,B 0,C 180,E1 -14463.717,E2 -14463.717} C_VEL
LIN {X 0,Y 338.74,Z 445.23,A -85,B 0,C 180,E1 -14464.595,E2 -14464.595} C_VEL
LIN {X 0,Y 341.573,Z 458.015,A -85,B 0,C 180,E1 -14465.569,E2 -14465.569} C_VEL
LIN {X 0,Y 343.552,Z 470.831,A -85,B 0,C 180,E1 -14466.701,E2 -14466.701} C_VEL
LIN {X 0,Y 342.138,Z 483.832,A -85,B 0,C 180,E1 -14467.873,E2 -14467.873} C_VEL
LIN {X 0,Y 340.309,Z 496.455,A -85,B 0,C 180,E1 -14469.288,E2 -14469.288} C_VEL
LIN {X 0,Y 338.462,Z 508.09,A -85,B 0,C 180,E1 -14470.911,E2 -14470.911} C_VEL
LIN {X 0,Y 336.788,Z 518.495,A -85,B 0,C 180,E1 -14472.7,E2 -14472.7} C_VEL
LIN {X 0,Y 335.343,Z 527.46,A -85,B 0,C 180,E1 -14474.591,E2 -14474.591} C_VEL
LIN {X 0,Y 334.263,Z 535.301,A -85,B 0,C 180,E1 -14476.627,E2 -14476.627} C_VEL
LIN {X 0,Y 333.296,Z 541.056,A -85,B 0,C 180,E1 -14478.444,E2 -14478.444} C_VEL
LIN {X 0,Y 332.735,Z 545.771,A -85,B 0,C 180,E1 -14480.272,E2 -14480.272} C_VEL
LIN {X 0,Y 332.198,Z 550.656,A -85,B 0,C 180,E1 -14482.707,E2 -14482.707} C_VEL
LIN {X 0,Y 331.974,Z 554.053,A -85,B 0,C 180,E1 -14485.142,E2 -14485.142} C_VEL
LIN {X 0,Y 331.881,Z 556.061,A -85,B 0,C 180,E1 -14487.573,E2 -14487.573} C_VEL
LIN {X 0,Y 331.883,Z 556.724,A -85,B 0,C 180,E1 -14490,E2 -14490} C_VEL
LIN {X 0,Y 331.881,Z 556.054,A -85,B 0,C 180,E1 -14492.427,E2 -14492.427} C_VEL
LIN {X 0,Y 331.977,Z 554.041,A -85,B 0,C 180,E1 -14494.858,E2 -14494.858} C_VEL
LIN {X 0,Y 332.238,Z 550.636,A -85,B 0,C 180,E1 -14497.292,E2 -14497.292} C_VEL
LIN {X 0,Y 332.723,Z 545.737,A -85,B 0,C 180,E1 -14499.728,E2 -14499.728} C_VEL
LIN {X 0,Y 333.57,Z 539.2,A -85,B 0,C 180,E1 -14502.163,E2 -14502.163} C_VEL
LIN {X 0,Y 334.547,Z 533.046,A -85,B 0,C 180,E1 -14503.98,E2 -14503.98} C_VEL
LIN {X 0,Y 335.854,Z 524.304,A -85,B 0,C 180,E1 -14506.097,E2 -14506.097} C_VEL
LIN {X 0,Y 337.344,Z 515.158,A -85,B 0,C 180,E1 -14507.896,E2 -14507.896} C_VEL
LIN {X 0,Y 339.139,Z 504.066,A -85,B 0,C 180,E1 -14509.679,E2 -14509.679} C_VEL
LIN {X 0,Y 340.883,Z 492.74,A -85,B 0,C 180,E1 -14511.149,E2 -14511.149} C_VEL
LIN {X 0,Y 342.47,Z 480.786,A -85,B 0,C 180,E1 -14512.413,E2 -14512.413} C_VEL
LIN {X 0,Y 343.475,Z 470.702,A -85,B 0,C 180,E1 -14513.299,E2 -14513.299} C_VEL
LIN {X 0,Y 341.541,Z 457.959,A -85,B 0,C 180,E1 -14514.419,E2 -14514.419} C_VEL
LIN {X 0,Y 338.524,Z 444.424,A -85,B 0,C 180,E1 -14515.446,E2 -14515.446} C_VEL
LIN {X 0,Y 334.693,Z 431.334,A -85,B 0,C 180,E1 -14516.298,E2 -14516.298} C_VEL
LIN {X 0,Y 333.144,Z 425.87,A -85,B 0,C 180,E1 -14516.606,E2 -14516.606} C_VEL
LIN {X 0,Y 333.609,Z 420.797,A -85,B 0,C 180,E1 -14520.371,E2 -14520.371} C_VEL
LIN {X 0,Y 333.986,Z 417.147,A -85,B 0,C 180,E1 -14523.169,E2 -14523.169} C_VEL
LIN {X 0,Y 334.385,Z 413.492,A -85,B 0,C 180,E1 -14526.05,E2 -14526.05} C_VEL
LIN {X 0,Y 334.632,Z 409.86,A -85,B 0,C 180,E1 -14529.055,E2 -14529.055} C_VEL
LIN {X 0,Y 334.394,Z 406.214,A -85,B 0,C 180,E1 -14532.264,E2 -14532.264} C_VEL
LIN {X 0,Y 333.811,Z 402.28,A -85,B 0,C 180,E1 -14535.991,E2 -14535.991} C_VEL
LIN {X 0,Y 333.687,Z 401.55,A -85,B 0,C 180,E1 -14536.786,E2 -14536.786} C_VEL
LIN {X 0,Y 333.673,Z 401.548,A -85,B 0,C 180,E1 -14540.811,E2 -14540.811} C_VEL
LIN {X 0,Y 333.678,Z 401.548,A -85,B 0,C 180,E1 -14543.861,E2 -14543.861} C_VEL
LIN {X 0,Y 333.646,Z 401.553,A -85,B 0,C 180,E1 -14547.412,E2 -14547.412} C_VEL
LIN {X 0,Y 333.691,Z 401.547,A -85,B 0,C 180,E1 -14551.026,E2 -14551.026} C_VEL
LIN {X 0,Y 333.735,Z 401.54,A -85,B 0,C 180,E1 -14553.754,E2 -14553.754} C_VEL
LIN {X 0,Y 333.657,Z 401.549,A -85,B 0,C 180,E1 -14557.719,E2 -14557.719} C_VEL
LIN {X 0,Y 333.796,Z 401.53,A -85,B 0,C 180,E1 -14561.59,E2 -14561.59} C_VEL
LIN {X 0,Y 333.809,Z 401.527,A -85,B 0,C 180,E1 -14565.577,E2 -14565.577} C_VEL
LIN {X 0,Y 333.835,Z 401.523,A -85,B 0,C 180,E1 -14569.078,E2 -14569.078} C_VEL
LIN {X 0,Y 334.027,Z 401.497,A -85,B 0,C 180,E1 -14572.748,E2 -14572.748} C_VEL
LIN {X 0,Y 333.813,Z 401.531,A -85,B 0,C 180,E1 -14575.169,E2 -14575.169} C_VEL
LIN {X 0,Y 334.109,Z 401.491,A -85,B 0,C 180,E1 -14577.589,E2 -14577.589} C_VEL
LIN {X 0,Y 334.268,Z 401.473,A -85,B 0,C 180,E1 -14580,E2 -14580} C_VEL
LIN {X 0,Y 334.107,Z 401.491,A -85,B 0,C 180,E1 -14582.411,E2 -14582.411} C_VEL
LIN {X 0,Y 334.027,Z 401.502,A -85,B 0,C 180,E1 -14587.253,E2 -14587.253} C_VEL
LIN {X 0,Y 333.836,Z 401.525,A -85,B 0,C 180,E1 -14590.922,E2 -14590.922} C_VEL
LIN {X 0,Y 333.81,Z 401.529,A -85,B 0,C 180,E1 -14594.634,E2 -14594.634} C_VEL
LIN {X 0,Y 333.798,Z 401.53,A -85,B 0,C 180,E1 -14598.656,E2 -14598.656} C_VEL
LIN {X 0,Y 333.693,Z 401.544,A -85,B 0,C 180,E1 -14602.278,E2 -14602.278} C_VEL
LIN {X 0,Y 333.736,Z 401.54,A -85,B 0,C 180,E1 -14606.246,E2 -14606.246} C_VEL
LIN {X 0,Y 333.691,Z 401.545,A -85,B 0,C 180,E1 -14608.974,E2 -14608.974} C_VEL
LIN {X 0,Y 333.647,Z 401.552,A -85,B 0,C 180,E1 -14612.588,E2 -14612.588} C_VEL
LIN {X 0,Y 333.679,Z 401.547,A -85,B 0,C 180,E1 -14616.139,E2 -14616.139} C_VEL
LIN {X 0,Y 333.648,Z 401.551,A -85,B 0,C 180,E1 -14619.192,E2 -14619.192} C_VEL
LIN {X 0,Y 333.634,Z 401.552,A -85,B 0,C 180,E1 -14622.5,E2 -14622.5} C_VEL
LIN {X 0,Y 333.639,Z 401.551,A -85,B 0,C 180,E1 -14625.962,E2 -14625.962} C_VEL
LIN {X 0,Y 334.081,Z 404.716,A -85,B 0,C 180,E1 -14629.297,E2 -14629.297} C_VEL
LIN {X 0,Y 334.051,Z 407.942,A -85,B 0,C 180,E1 -14632.402,E2 -14632.402} C_VEL
LIN {X 0,Y 333.902,Z 411.133,A -85,B 0,C 180,E1 -14635.368,E2 -14635.368} C_VEL
LIN {X 0,Y 333.572,Z 414.36,A -85,B 0,C 180,E1 -14638.216,E2 -14638.216} C_VEL
LIN {X 0,Y 333.323,Z 417.584,A -85,B 0,C 180,E1 -14640.991,E2 -14640.991} C_VEL
LIN {X 0,Y 333.11,Z 420.487,A -85,B 0,C 180,E1 -14643.448,E2 -14643.448} C_VEL
LIN {X 0,Y 334.916,Z 426.311,A -85,B 0,C 180,E1 -14643.795,E2 -14643.795} C_VEL
LIN {X 0,Y 339.144,Z 440.307,A -85,B 0,C 180,E1 -14644.746,E2 -14644.746} C_VEL
LIN {X 0,Y 342.09,Z 452.922,A -85,B 0,C 180,E1 -14645.74,E2 -14645.74} C_VEL
LIN {X 0,Y 343.924,Z 464.338,A -85,B 0,C 180,E1 -14646.756,E2 -14646.756} C_VEL
LIN {X 0,Y 342.5,Z 477.133,A -85,B 0,C 180,E1 -14647.897,E2 -14647.897} C_VEL
LIN {X 0,Y 340.875,Z 488.652,A -85,B 0,C 180,E1 -14649.167,E2 -14649.167} C_VEL
LIN {X 0,Y 339.093,Z 499.558,A -85,B 0,C 180,E1 -14650.633,E2 -14650.633} C_VEL
LIN {X 0,Y 337.658,Z 508.693,A -85,B 0,C 180,E1 -14652.121,E2 -14652.121} C_VEL
LIN {X 0,Y 336.154,Z 517.845,A -85,B 0,C 180,E1 -14653.918,E2 -14653.918} C_VEL
LIN {X 0,Y 334.887,Z 526.582,A -85,B 0,C 180,E1 -14656.034,E2 -14656.034} C_VEL
LIN {X 0,Y 333.78,Z 532.74,A -85,B 0,C 180,E1 -14657.845,E2 -14657.845} C_VEL
LIN {X 0,Y 333.11,Z 537.827,A -85,B 0,C 180,E1 -14659.669,E2 -14659.669} C_VEL
LIN {X 0,Y 332.441,Z 543.102,A -85,B 0,C 180,E1 -14662.102,E2 -14662.102} C_VEL
LIN {X 0,Y 332.221,Z 546.044,A -85,B 0,C 180,E1 -14663.928,E2 -14663.928} C_VEL
LIN {X 0,Y 332.017,Z 548.748,A -85,B 0,C 180,E1 -14666.359,E2 -14666.359} C_VEL
LIN {X 0,Y 331.875,Z 550.102,A -85,B 0,C 180,E1 -14668.787,E2 -14668.787} C_VEL
LIN {X 0,Y 331.875,Z 550.134,A -85,B 0,C 180,E1 -14671.214,E2 -14671.214} C_VEL
LIN {X 0,Y 332.016,Z 548.84,A -85,B 0,C 180,E1 -14673.641,E2 -14673.641} C_VEL
LIN {X 0,Y 332.219,Z 546.101,A -85,B 0,C 180,E1 -14676.133,E2 -14676.133} C_VEL
LIN {X 0,Y 332.57,Z 542.12,A -85,B 0,C 180,E1 -14678.507,E2 -14678.507} C_VEL
LIN {X 0,Y 333.313,Z 536.494,A -85,B 0,C 180,E1 -14680.939,E2 -14680.939} C_VEL
LIN {X 0,Y 334.305,Z 530.141,A -85,B 0,C 180,E1 -14683.062,E2 -14683.062} C_VEL
LIN {X 0,Y 335.395,Z 522.917,A -85,B 0,C 180,E1 -14685.014,E2 -14685.014} C_VEL
LIN {X 0,Y 336.815,Z 513.981,A -85,B 0,C 180,E1 -14686.985,E2 -14686.985} C_VEL
LIN {X 0,Y 338.44,Z 504.024,A -85,B 0,C 180,E1 -14688.776,E2 -14688.776} C_VEL
LIN {X 0,Y 340.251,Z 492.938,A -85,B 0,C 180,E1 -14690.399,E2 -14690.399} C_VEL
LIN {X 0,Y 342.047,Z 480.67,A -85,B 0,C 180,E1 -14691.845,E2 -14691.845} C_VEL
LIN {X 0,Y 343.502,Z 468.861,A -85,B 0,C 180,E1 -14692.972,E2 -14692.972} C_VEL
LIN {X 0,Y 343.925,Z 463.341,A -85,B 0,C 180,E1 -14693.435,E2 -14693.435} C_VEL
LIN {X 0,Y 341.77,Z 451.375,A -85,B 0,C 180,E1 -14694.503,E2 -14694.503} C_VEL
LIN {X 0,Y 338.548,Z 438.067,A -85,B 0,C 180,E1 -14695.528,E2 -14695.528} C_VEL
LIN {X 0,Y 334.045,Z 423.66,A -85,B 0,C 180,E1 -14696.473,E2 -14696.473} C_VEL
LIN {X 0,Y 333.107,Z 420.451,A -85,B 0,C 180,E1 -14696.68,E2 -14696.68} C_VEL
LIN {X 0,Y 333.4,Z 416.082,A -85,B 0,C 180,E1 -14700.392,E2 -14700.392} C_VEL
LIN {X 0,Y 333.701,Z 412.876,A -85,B 0,C 180,E1 -14703.201,E2 -14703.201} C_VEL
LIN {X 0,Y 333.988,Z 409.672,A -85,B 0,C 180,E1 -14706.1,E2 -14706.1} C_VEL
LIN {X 0,Y 334.116,Z 406.434,A -85,B 0,C 180,E1 -14709.127,E2 -14709.127} C_VEL
LIN {X 0,Y 334.086,Z 404.749,A -85,B 0,C 180,E1 -14710.772,E2 -14710.772} C_VEL
LIN {X 0,Y 333.661,Z 401.606,A -85,B 0,C 180,E1 -14714.035,E2 -14714.035} C_VEL
LIN {X 0,Y 333.644,Z 401.556,A -85,B 0,C 180,E1 -14717.619,E2 -14717.619} C_VEL
LIN {X 0,Y 333.655,Z 401.551,A -85,B 0,C 180,E1 -14721.202,E2 -14721.202} C_VEL
LIN {X 0,Y 333.65,Z 401.549,A -85,B 0,C 180,E1 -14722.251,E2 -14722.251} C_VEL
LIN {X 0,Y 333.031,Z 401.63,A -85,B 0,C 180,E1 -14723.259,E2 -14723.259} C_VEL
LIN {X 0,Y 330.214,Z 401.986,A -85,B 0,C 180,E1 -14724.898,E2 -14724.898} C_VEL
LIN {X 0,Y 327.781,Z 402.288,A -85,B 0,C 180,E1 -14726.226,E2 -14726.226} C_VEL
LIN {X 0,Y 326.704,Z 402.417,A -85,B 0,C 180,E1 -14727.254,E2 -14727.254} C_VEL
LIN {X 0,Y 326.601,Z 402.427,A -85,B 0,C 180,E1 -14727.602,E2 -14727.602} C_VEL
LIN {X 0,Y 326.663,Z 402.418,A -85,B 0,C 180,E1 -14730.341,E2 -14730.341} C_VEL
LIN {X 0,Y 326.692,Z 402.417,A -85,B 0,C 180,E1 -14734.516,E2 -14734.516} C_VEL
LIN {X 0,Y 326.652,Z 402.422,A -85,B 0,C 180,E1 -14738.546,E2 -14738.546} C_VEL
LIN {X 0,Y 326.747,Z 402.409,A -85,B 0,C 180,E1 -14741.177,E2 -14741.177} C_VEL
LIN {X 0,Y 326.766,Z 402.409,A -85,B 0,C 180,E1 -14745.433,E2 -14745.433} C_VEL
LIN {X 0,Y 326.773,Z 402.406,A -85,B 0,C 180,E1 -14748.839,E2 -14748.839} C_VEL
LIN {X 0,Y 326.982,Z 402.379,A -85,B 0,C 180,E1 -14752.59,E2 -14752.59} C_VEL
LIN {X 0,Y 326.781,Z 402.407,A -85,B 0,C 180,E1 -14755.065,E2 -14755.065} C_VEL
LIN {X 0,Y 327.049,Z 402.371,A -85,B 0,C 180,E1 -14757.537,E2 -14757.537} C_VEL
LIN {X 0,Y 327.2,Z 402.355,A -85,B 0,C 180,E1 -14760,E2 -14760} C_VEL
LIN {X 0,Y 327.051,Z 402.371,A -85,B 0,C 180,E1 -14762.463,E2 -14762.463} C_VEL
LIN {X 0,Y 326.999,Z 402.377,A -85,B 0,C 180,E1 -14766.169,E2 -14766.169} C_VEL
LIN {X 0,Y 326.917,Z 402.388,A -85,B 0,C 180,E1 -14768.655,E2 -14768.655} C_VEL
LIN {X 0,Y 326.738,Z 402.41,A -85,B 0,C 180,E1 -14772.421,E2 -14772.421} C_VEL
LIN {X 0,Y 326.756,Z 402.409,A -85,B 0,C 180,E1 -14774.957,E2 -14774.957} C_VEL
LIN {X 0,Y 326.736,Z 402.41,A -85,B 0,C 180,E1 -14778.839,E2 -14778.839} C_VEL
LIN {X 0,Y 326.623,Z 402.424,A -85,B 0,C 180,E1 -14782.787,E2 -14782.787} C_VEL
LIN {X 0,Y 326.692,Z 402.416,A -85,B 0,C 180,E1 -14785.484,E2 -14785.484} C_VEL
LIN {X 0,Y 326.649,Z 402.418,A -85,B 0,C 180,E1 -14789.66,E2 -14789.66} C_VEL
LIN {X 0,Y 326.62,Z 402.427,A -85,B 0,C 180,E1 -14792.946,E2 -14792.946} C_VEL
LIN {X 0,Y 326.615,Z 402.429,A -85,B 0,C 180,E1 -14795.519,E2 -14795.519} C_VEL
LIN {X 0,Y 326.637,Z 402.428,A -85,B 0,C 180,E1 -14799.232,E2 -14799.232} C_VEL
LIN {X 0,Y 326.652,Z 402.556,A -85,B 0,C 180,E1 -14802.986,E2 -14802.986} C_VEL
LIN {X 0,Y 327.216,Z 406.183,A -85,B 0,C 180,E1 -14806.583,E2 -14806.583} C_VEL
LIN {X 0,Y 327.563,Z 409.828,A -85,B 0,C 180,E1 -14809.934,E2 -14809.934} C_VEL
LIN {X 0,Y 327.461,Z 413.464,A -85,B 0,C 180,E1 -14813.063,E2 -14813.063} C_VEL
LIN {X 0,Y 327.055,Z 417.104,A -85,B 0,C 180,E1 -14816.033,E2 -14816.033} C_VEL
LIN {X 0,Y 326.593,Z 421.397,A -85,B 0,C 180,E1 -14819.403,E2 -14819.403} C_VEL
LIN {X 0,Y 326.201,Z 425.821,A -85,B 0,C 180,E1 -14822.781,E2 -14822.781} C_VEL
LIN {X 0,Y 327.888,Z 431.632,A -85,B 0,C 180,E1 -14823.106,E2 -14823.106} C_VEL
LIN {X 0,Y 332.057,Z 445.879,A -85,B 0,C 180,E1 -14824.085,E2 -14824.085} C_VEL
LIN {X 0,Y 335.049,Z 459.783,A -85,B 0,C 180,E1 -14825.195,E2 -14825.195} C_VEL
LIN {X 0,Y 336.899,Z 472.528,A -85,B 0,C 180,E1 -14826.376,E2 -14826.376} C_VEL
LIN {X 0,Y 335.261,Z 485.908,A -85,B 0,C 180,E1 -14827.638,E2 -14827.638} C_VEL
LIN {X 0,Y 333.468,Z 497.564,A -85,B 0,C 180,E1 -14829.005,E2 -14829.005} C_VEL
LIN {X 0,Y 331.744,Z 508.023,A -85,B 0,C 180,E1 -14830.509,E2 -14830.509} C_VEL
LIN {X 0,Y 329.977,Z 518.428,A -85,B 0,C 180,E1 -14832.332,E2 -14832.332} C_VEL
LIN {X 0,Y 328.361,Z 527.946,A -85,B 0,C 180,E1 -14834.396,E2 -14834.396} C_VEL
LIN {X 0,Y 327.132,Z 536.243,A -85,B 0,C 180,E1 -14836.647,E2 -14836.647} C_VEL
LIN {X 0,Y 326.059,Z 542.655,A -85,B 0,C 180,E1 -14838.814,E2 -14838.814} C_VEL
LIN {X 0,Y 325.388,Z 548.34,A -85,B 0,C 180,E1 -14841.304,E2 -14841.304} C_VEL
LIN {X 0,Y 325.008,Z 552.465,A -85,B 0,C 180,E1 -14843.793,E2 -14843.793} C_VEL
LIN {X 0,Y 324.858,Z 555.158,A -85,B 0,C 180,E1 -14846.279,E2 -14846.279} C_VEL
LIN {X 0,Y 324.774,Z 556.491,A -85,B 0,C 180,E1 -14848.76,E2 -14848.76} C_VEL
LIN {X 0,Y 324.774,Z 556.487,A -85,B 0,C 180,E1 -14851.24,E2 -14851.24} C_VEL
LIN {X 0,Y 324.858,Z 555.148,A -85,B 0,C 180,E1 -14853.721,E2 -14853.721} C_VEL
LIN {X 0,Y 325.009,Z 552.448,A -85,B 0,C 180,E1 -14856.207,E2 -14856.207} C_VEL
LIN {X 0,Y 325.377,Z 548.311,A -85,B 0,C 180,E1 -14858.696,E2 -14858.696} C_VEL
LIN {X 0,Y 326.057,Z 542.614,A -85,B 0,C 180,E1 -14861.186,E2 -14861.186} C_VEL
LIN {X 0,Y 327.128,Z 536.194,A -85,B 0,C 180,E1 -14863.353,E2 -14863.353} C_VEL
LIN {X 0,Y 328.37,Z 527.862,A -85,B 0,C 180,E1 -14865.609,E2 -14865.609} C_VEL
LIN {X 0,Y 329.97,Z 518.345,A -85,B 0,C 180,E1 -14867.668,E2 -14867.668} C_VEL
LIN {X 0,Y 331.759,Z 507.922,A -85,B 0,C 180,E1 -14869.49,E2 -14869.49} C_VEL
LIN {X 0,Y 333.658,Z 496.265,A -85,B 0,C 180,E1 -14871.144,E2 -14871.144} C_VEL
LIN {X 0,Y 335.46,Z 484.153,A -85,B 0,C 180,E1 -14872.531,E2 -14872.531} C_VEL
LIN {X 0,Y 336.845,Z 472.369,A -85,B 0,C 180,E1 -14873.625,E2 -14873.625} C_VEL
LIN {X 0,Y 335.004,Z 459.52,A -85,B 0,C 180,E1 -14874.808,E2 -14874.808} C_VEL
LIN {X 0,Y 332.016,Z 445.784,A -85,B 0,C 180,E1 -14875.903,E2 -14875.903} C_VEL
LIN {X 0,Y 327.946,Z 431.761,A -85,B 0,C 180,E1 -14876.863,E2 -14876.863} C_VEL
LIN {X 0,Y 326.184,Z 425.794,A -85,B 0,C 180,E1 -14877.22,E2 -14877.22} C_VEL
LIN {X 0,Y 326.636,Z 420.733,A -85,B 0,C 180,E1 -14881.09,E2 -14881.09} C_VEL
LIN {X 0,Y 327.054,Z 417.075,A -85,B 0,C 180,E1 -14883.967,E2 -14883.967} C_VEL
LIN {X 0,Y 327.5,Z 412.846,A -85,B 0,C 180,E1 -14887.439,E2 -14887.439} C_VEL
LIN {X 0,Y 327.56,Z 409.795,A -85,B 0,C 180,E1 -14890.066,E2 -14890.066} C_VEL
LIN {X 0,Y 327.196,Z 406.149,A -85,B 0,C 180,E1 -14893.42,E2 -14893.42} C_VEL
LIN {X 0,Y 326.632,Z 402.429,A -85,B 0,C 180,E1 -14897.116,E2 -14897.116} C_VEL
LIN {X 0,Y 326.645,Z 402.424,A -85,B 0,C 180,E1 -14901.394,E2 -14901.394} C_VEL
LIN {X 0,Y 326.621,Z 402.427,A -85,B 0,C 180,E1 -14904.851,E2 -14904.851} C_VEL
LIN {X 0,Y 326.61,Z 402.43,A -85,B 0,C 180,E1 -14907.456,E2 -14907.456} C_VEL
LIN {X 0,Y 326.648,Z 402.423,A -85,B 0,C 180,E1 -14910.34,E2 -14910.34} C_VEL
LIN {X 0,Y 326.69,Z 402.417,A -85,B 0,C 180,E1 -14914.516,E2 -14914.516} C_VEL
LIN {X 0,Y 326.621,Z 402.425,A -85,B 0,C 180,E1 -14918.544,E2 -14918.544} C_VEL
LIN {X 0,Y 326.745,Z 402.409,A -85,B 0,C 180,E1 -14921.178,E2 -14921.178} C_VEL
LIN {X 0,Y 326.764,Z 402.405,A -85,B 0,C 180,E1 -14925.433,E2 -14925.433} C_VEL
LIN {X 0,Y 326.771,Z 402.403,A -85,B 0,C 180,E1 -14928.839,E2 -14928.839} C_VEL
LIN {X 0,Y 326.981,Z 402.374,A -85,B 0,C 180,E1 -14932.59,E2 -14932.59} C_VEL
LIN {X 0,Y 326.78,Z 402.407,A -85,B 0,C 180,E1 -14935.065,E2 -14935.065} C_VEL
LIN {X 0,Y 327.049,Z 402.37,A -85,B 0,C 180,E1 -14937.537,E2 -14937.537} C_VEL
LIN {X 0,Y 327.219,Z 402.351,A -85,B 0,C 180,E1 -14940,E2 -14940} C_VEL
LIN {X 0,Y 327.047,Z 402.37,A -85,B 0,C 180,E1 -14942.463,E2 -14942.463} C_VEL
LIN {X 0,Y 326.972,Z 402.379,A -85,B 0,C 180,E1 -14946.677,E2 -14946.677} C_VEL
LIN {X 0,Y 326.816,Z 402.401,A -85,B 0,C 180,E1 -14949.906,E2 -14949.906} C_VEL
LIN {X 0,Y 326.76,Z 402.403,A -85,B 0,C 180,E1 -14953.685,E2 -14953.685} C_VEL
LIN {X 0,Y 326.702,Z 402.411,A -85,B 0,C 180,E1 -14957.528,E2 -14957.528} C_VEL
LIN {X 0,Y 326.669,Z 402.418,A -85,B 0,C 180,E1 -14960.135,E2 -14960.135} C_VEL
LIN {X 0,Y 326.653,Z 402.422,A -85,B 0,C 180,E1 -14964.129,E2 -14964.129} C_VEL
LIN {X 0,Y 326.684,Z 402.417,A -85,B 0,C 180,E1 -14966.858,E2 -14966.858} C_VEL
LIN {X 0,Y 326.635,Z 402.424,A -85,B 0,C 180,E1 -14970.61,E2 -14970.61} C_VEL
LIN {X 0,Y 326.609,Z 402.428,A -85,B 0,C 180,E1 -14974.019,E2 -14974.019} C_VEL
LIN {X 0,Y 326.631,Z 402.426,A -85,B 0,C 180,E1 -14977.239,E2 -14977.239} C_VEL
LIN {X 0,Y 326.579,Z 402.43,A -85,B 0,C 180,E1 -14981.131,E2 -14981.131} C_VEL
LIN {X 0,Y 326.562,Z 402.434,A -85,B 0,C 180,E1 -14984.749,E2 -14984.749} C_VEL
LIN {X 0,Y 326.566,Z 402.433,A -85,B 0,C 180,E1 -14985.251,E2 -14985.251} C_VEL
LIN {X 0,Y 326.782,Z 403.613,A -85,B 0,C 180,E1 -14986.99,E2 -14986.99} C_VEL
LIN {X 0,Y 327.062,Z 406.38,A -85,B 0,C 180,E1 -14989.861,E2 -14989.861} C_VEL
LIN {X 0,Y 327.006,Z 409.621,A -85,B 0,C 180,E1 -14993.003,E2 -14993.003} C_VEL
LIN {X 0,Y 326.753,Z 412.815,A -85,B 0,C 180,E1 -14995.998,E2 -14995.998} C_VEL
LIN {X 0,Y 326.389,Z 416.67,A -85,B 0,C 180,E1 -14999.464,E2 -14999.464} C_VEL
LIN {X 0,Y 326.123,Z 420.573,A -85,B 0,C 180,E1 -15002.841,E2 -15002.841} C_VEL
LIN {X 0,Y 328.972,Z 429.46,A -85,B 0,C 180,E1 -15003.4,E2 -15003.4} C_VEL
LIN {X 0,Y 332.953,Z 443.18,A -85,B 0,C 180,E1 -15004.397,E2 -15004.397} C_VEL
LIN {X 0,Y 335.893,Z 456.315,A -85,B 0,C 180,E1 -15005.505,E2 -15005.505} C_VEL
LIN {X 0,Y 337.222,Z 464.653,A -85,B 0,C 180,E1 -15006.288,E2 -15006.288} C_VEL
LIN {X 0,Y 335.907,Z 477.419,A -85,B 0,C 180,E1 -15007.464,E2 -15007.464} C_VEL
LIN {X 0,Y 334.24,Z 488.725,A -85,B 0,C 180,E1 -15008.733,E2 -15008.733} C_VEL
LIN {X 0,Y 332.385,Z 499.631,A -85,B 0,C 180,E1 -15010.226,E2 -15010.226} C_VEL
LIN {X 0,Y 330.588,Z 510.389,A -85,B 0,C 180,E1 -15012.046,E2 -15012.046} C_VEL
LIN {X 0,Y 328.947,Z 519.954,A -85,B 0,C 180,E1 -15014.036,E2 -15014.036} C_VEL
LIN {X 0,Y 327.771,Z 527.767,A -85,B 0,C 180,E1 -15016.042,E2 -15016.042} C_VEL
LIN {X 0,Y 326.563,Z 534.614,A -85,B 0,C 180,E1 -15018.203,E2 -15018.203} C_VEL
LIN {X 0,Y 325.881,Z 539.339,A -85,B 0,C 180,E1 -15020.065,E2 -15020.065} C_VEL
LIN {X 0,Y 325.301,Z 544.233,A -85,B 0,C 180,E1 -15022.552,E2 -15022.552} C_VEL
LIN {X 0,Y 324.996,Z 547.638,A -85,B 0,C 180,E1 -15025.038,E2 -15025.038} C_VEL
LIN {X 0,Y 324.838,Z 549.66,A -85,B 0,C 180,E1 -15027.52,E2 -15027.52} C_VEL
LIN {X 0,Y 324.793,Z 550.352,A -85,B 0,C 180,E1 -15030,E2 -15030} C_VEL
LIN {X 0,Y 324.837,Z 549.722,A -85,B 0,C 180,E1 -15032.48,E2 -15032.48} C_VEL
LIN {X 0,Y 324.995,Z 547.756,A -85,B 0,C 180,E1 -15034.962,E2 -15034.962} C_VEL
LIN {X 0,Y 325.291,Z 544.408,A -85,B 0,C 180,E1 -15037.448,E2 -15037.448} C_VEL
LIN {X 0,Y 325.853,Z 539.579,A -85,B 0,C 180,E1 -15039.936,E2 -15039.936} C_VEL
LIN {X 0,Y 326.533,Z 534.918,A -85,B 0,C 180,E1 -15041.799,E2 -15041.799} C_VEL
LIN {X 0,Y 327.735,Z 528.138,A -85,B 0,C 180,E1 -15043.96,E2 -15043.96} C_VEL
LIN {X 0,Y 329.067,Z 519.718,A -85,B 0,C 180,E1 -15046.12,E2 -15046.12} C_VEL
LIN {X 0,Y 330.548,Z 510.93,A -85,B 0,C 180,E1 -15047.957,E2 -15047.957} C_VEL
LIN {X 0,Y 332.368,Z 500.278,A -85,B 0,C 180,E1 -15049.775,E2 -15049.775} C_VEL
LIN {X 0,Y 334.143,Z 489.503,A -85,B 0,C 180,E1 -15051.274,E2 -15051.274} C_VEL
LIN {X 0,Y 335.923,Z 477.356,A -85,B 0,C 180,E1 -15052.649,E2 -15052.649} C_VEL
LIN {X 0,Y 337.284,Z 465.947,A -85,B 0,C 180,E1 -15053.695,E2 -15053.695} C_VEL
LIN {X 0,Y 336.145,Z 457.689,A -85,B 0,C 180,E1 -15054.483,E2 -15054.483} C_VEL
LIN {X 0,Y 333.285,Z 444.366,A -85,B 0,C 180,E1 -15055.621,E2 -15055.621} C_VEL
LIN {X 0,Y 329.282,Z 430.515,A -85,B 0,C 180,E1 -15056.644,E2 -15056.644} C_VEL
LIN {X 0,Y 326.124,Z 420.538,A -85,B 0,C 180,E1 -15057.288,E2 -15057.288} C_VEL
LIN {X 0,Y 326.417,Z 416.16,A -85,B 0,C 180,E1 -15061.114,E2 -15061.114} C_VEL
LIN {X 0,Y 326.744,Z 412.955,A -85,B 0,C 180,E1 -15064.003,E2 -15064.003} C_VEL
LIN {X 0,Y 327.009,Z 409.367,A -85,B 0,C 180,E1 -15067.326,E2 -15067.326} C_VEL
LIN {X 0,Y 327.064,Z 406.495,A -85,B 0,C 180,E1 -15070.139,E2 -15070.139} C_VEL
LIN {X 0,Y 326.724,Z 403.271,A -85,B 0,C 180,E1 -15073.499,E2 -15073.499} C_VEL
LIN {X 0,Y 326.575,Z 402.436,A -85,B 0,C 180,E1 -15074.751,E2 -15074.751} C_VEL
LIN {X 0,Y 326.578,Z 402.435,A -85,B 0,C 180,E1 -15078.154,E2 -15078.154} C_VEL
LIN {X 0,Y 326.626,Z 402.426,A -85,B 0,C 180,E1 -15081.392,E2 -15081.392} C_VEL
LIN {X 0,Y 326.622,Z 402.426,A -85,B 0,C 180,E1 -15084.851,E2 -15084.851} C_VEL
LIN {X 0,Y 326.601,Z 402.427,A -85,B 0,C 180,E1 -15087.602,E2 -15087.602} C_VEL
LIN {X 0,Y 325.897,Z 402.515,A -85,B 0,C 180,E1 -15088.632,E2 -15088.632} C_VEL
LIN {X 0,Y 323.057,Z 402.868,A -85,B 0,C 180,E1 -15090.309,E2 -15090.309} C_VEL
LIN {X 0,Y 320.683,Z 403.164,A -85,B 0,C 180,E1 -15091.668,E2 -15091.668} C_VEL
LIN {X 0,Y 319.675,Z 403.292,A -85,B 0,C 180,E1 -15092.719,E2 -15092.719} C_VEL
LIN {X 0,Y 319.598,Z 403.298,A -85,B 0,C 180,E1 -15093.075,E2 -15093.075} C_VEL
LIN {X 0,Y 319.573,Z 403.299,A -85,B 0,C 180,E1 -15096.681,E2 -15096.681} C_VEL
LIN {X 0,Y 319.692,Z 403.289,A -85,B 0,C 180,E1 -15100.962,E2 -15100.962} C_VEL
LIN {X 0,Y 319.733,Z 403.284,A -85,B 0,C 180,E1 -15105.276,E2 -15105.276} C_VEL
LIN {X 0,Y 319.761,Z 403.279,A -85,B 0,C 180,E1 -15109.873,E2 -15109.873} C_VEL
LIN {X 0,Y 319.936,Z 403.257,A -85,B 0,C 180,E1 -15112.426,E2 -15112.426} C_VEL
LIN {X 0,Y 319.75,Z 403.282,A -85,B 0,C 180,E1 -15114.956,E2 -15114.956} C_VEL
LIN {X 0,Y 319.992,Z 403.25,A -85,B 0,C 180,E1 -15117.482,E2 -15117.482} C_VEL
LIN {X 0,Y 320.152,Z 403.232,A -85,B 0,C 180,E1 -15120,E2 -15120} C_VEL
LIN {X 0,Y 319.994,Z 403.25,A -85,B 0,C 180,E1 -15122.517,E2 -15122.517} C_VEL
LIN {X 0,Y 319.955,Z 403.255,A -85,B 0,C 180,E1 -15126.305,E2 -15126.305} C_VEL
LIN {X 0,Y 319.845,Z 403.269,A -85,B 0,C 180,E1 -15128.848,E2 -15128.848} C_VEL
LIN {X 0,Y 319.685,Z 403.289,A -85,B 0,C 180,E1 -15132.7,E2 -15132.7} C_VEL
LIN {X 0,Y 319.702,Z 403.286,A -85,B 0,C 180,E1 -15135.295,E2 -15135.295} C_VEL
LIN {X 0,Y 319.678,Z 403.29,A -85,B 0,C 180,E1 -15139.255,E2 -15139.255} C_VEL
LIN {X 0,Y 319.572,Z 403.299,A -85,B 0,C 180,E1 -15143.319,E2 -15143.319} C_VEL
LIN {X 0,Y 319.636,Z 403.295,A -85,B 0,C 180,E1 -15146.088,E2 -15146.088} C_VEL
LIN {X 0,Y 319.582,Z 403.303,A -85,B 0,C 180,E1 -15148.934,E2 -15148.934} C_VEL
LIN {X 0,Y 319.533,Z 403.308,A -85,B 0,C 180,E1 -15151.862,E2 -15151.862} C_VEL
LIN {X 0,Y 319.582,Z 403.306,A -85,B 0,C 180,E1 -15155.543,E2 -15155.543} C_VEL
LIN {X 0,Y 319.601,Z 403.304,A -85,B 0,C 180,E1 -15158.004,E2 -15158.004} C_VEL
LIN {X 0,Y 319.619,Z 403.301,A -85,B 0,C 180,E1 -15162.435,E2 -15162.435} C_VEL
LIN {X 0,Y 320.19,Z 407.206,A -85,B 0,C 180,E1 -15166.413,E2 -15166.413} C_VEL
LIN {X 0,Y 320.471,Z 409.774,A -85,B 0,C 180,E1 -15168.859,E2 -15168.859} C_VEL
LIN {X 0,Y 320.569,Z 411.598,A -85,B 0,C 180,E1 -15170.522,E2 -15170.522} C_VEL
LIN {X 0,Y 320.322,Z 415.216,A -85,B 0,C 180,E1 -15173.673,E2 -15173.673} C_VEL
LIN {X 0,Y 319.933,Z 418.879,A -85,B 0,C 180,E1 -15176.689,E2 -15176.689} C_VEL
LIN {X 0,Y 319.511,Z 422.515,A -85,B 0,C 180,E1 -15179.608,E2 -15179.608} C_VEL
LIN {X 0,Y 319.208,Z 425.714,A -85,B 0,C 180,E1 -15182.103,E2 -15182.103} C_VEL
LIN {X 0,Y 324.343,Z 442.832,A -85,B 0,C 180,E1 -15183.265,E2 -15183.265} C_VEL
LIN {X 0,Y 327.517,Z 456.081,A -85,B 0,C 180,E1 -15184.323,E2 -15184.323} C_VEL
LIN {X 0,Y 329.576,Z 468.374,A -85,B 0,C 180,E1 -15185.447,E2 -15185.447} C_VEL
LIN {X 0,Y 330.243,Z 474.057,A -85,B 0,C 180,E1 -15186.02,E2 -15186.02} C_VEL
LIN {X 0,Y 328.659,Z 486.057,A -85,B 0,C 180,E1 -15187.189,E2 -15187.189} C_VEL
LIN {X 0,Y 326.627,Z 498.67,A -85,B 0,C 180,E1 -15188.709,E2 -15188.709} C_VEL
LIN {X 0,Y 324.692,Z 509.85,A -85,B 0,C 180,E1 -15190.397,E2 -15190.397} C_VEL
LIN {X 0,Y 322.899,Z 519.879,A -85,B 0,C 180,E1 -15192.259,E2 -15192.259} C_VEL
LIN {X 0,Y 321.384,Z 528.428,A -85,B 0,C 180,E1 -15194.194,E2 -15194.194} C_VEL
LIN {X 0,Y 320.197,Z 536.175,A -85,B 0,C 180,E1 -15196.352,E2 -15196.352} C_VEL
LIN {X 0,Y 319.047,Z 542.587,A -85,B 0,C 180,E1 -15198.565,E2 -15198.565} C_VEL
LIN {X 0,Y 318.348,Z 548.272,A -85,B 0,C 180,E1 -15201.11,E2 -15201.11} C_VEL
LIN {X 0,Y 317.917,Z 552.396,A -85,B 0,C 180,E1 -15203.654,E2 -15203.654} C_VEL
LIN {X 0,Y 317.769,Z 555.09,A -85,B 0,C 180,E1 -15206.195,E2 -15206.195} C_VEL
LIN {X 0,Y 317.689,Z 556.422,A -85,B 0,C 180,E1 -15208.732,E2 -15208.732} C_VEL
LIN {X 0,Y 317.689,Z 556.418,A -85,B 0,C 180,E1 -15211.267,E2 -15211.267} C_VEL
LIN {X 0,Y 317.77,Z 555.079,A -85,B 0,C 180,E1 -15213.804,E2 -15213.804} C_VEL
LIN {X 0,Y 317.921,Z 552.378,A -85,B 0,C 180,E1 -15216.346,E2 -15216.346} C_VEL
LIN {X 0,Y 318.336,Z 548.241,A -85,B 0,C 180,E1 -15218.89,E2 -15218.89} C_VEL
LIN {X 0,Y 319.045,Z 542.543,A -85,B 0,C 180,E1 -15221.435,E2 -15221.435} C_VEL
LIN {X 0,Y 320.195,Z 536.123,A -85,B 0,C 180,E1 -15223.648,E2 -15223.648} C_VEL
LIN {X 0,Y 321.392,Z 528.342,A -85,B 0,C 180,E1 -15225.811,E2 -15225.811} C_VEL
LIN {X 0,Y 322.896,Z 519.799,A -85,B 0,C 180,E1 -15227.741,E2 -15227.741} C_VEL
LIN {X 0,Y 324.705,Z 509.753,A -85,B 0,C 180,E1 -15229.602,E2 -15229.602} C_VEL
LIN {X 0,Y 326.623,Z 498.541,A -85,B 0,C 180,E1 -15231.291,E2 -15231.291} C_VEL
LIN {X 0,Y 328.632,Z 485.948,A -85,B 0,C 180,E1 -15232.808,E2 -15232.808} C_VEL
LIN {X 0,Y 330.185,Z 473.871,A -85,B 0,C 180,E1 -15233.983,E2 -15233.983} C_VEL
LIN {X 0,Y 328.615,Z 462.076,A -85,B 0,C 180,E1 -15235.127,E2 -15235.127} C_VEL
LIN {X 0,Y 326.049,Z 449.543,A -85,B 0,C 180,E1 -15236.197,E2 -15236.197} C_VEL
LIN {X 0,Y 322.52,Z 436.689,A -85,B 0,C 180,E1 -15237.16,E2 -15237.16} C_VEL
LIN {X 0,Y 319.199,Z 425.742,A -85,B 0,C 180,E1 -15237.853,E2 -15237.853} C_VEL
LIN {X 0,Y 319.674,Z 420.655,A -85,B 0,C 180,E1 -15241.846,E2 -15241.846} C_VEL
LIN {X 0,Y 320.143,Z 417.032,A -85,B 0,C 180,E1 -15244.804,E2 -15244.804} C_VEL
LIN {X 0,Y 320.483,Z 413.372,A -85,B 0,C 180,E1 -15247.881,E2 -15247.881} C_VEL
LIN {X 0,Y 320.548,Z 411.111,A -85,B 0,C 180,E1 -15249.881,E2 -15249.881} C_VEL
LIN {X 0,Y 320.262,Z 407.915,A -85,B 0,C 180,E1 -15252.865,E2 -15252.865} C_VEL
LIN {X 0,Y 319.776,Z 404.28,A -85,B 0,C 180,E1 -15256.491,E2 -15256.491} C_VEL
LIN {X 0,Y 319.584,Z 403.306,A -85,B 0,C 180,E1 -15257.768,E2 -15257.768} C_VEL
LIN {X 0,Y 319.599,Z 403.301,A -85,B 0,C 180,E1 -15261.996,E2 -15261.996} C_VEL
LIN {X 0,Y 319.561,Z 403.306,A -85,B 0,C 180,E1 -15265.124,E2 -15265.124} C_VEL
LIN {X 0,Y 319.567,Z 403.307,A -85,B 0,C 180,E1 -15269.059,E2 -15269.059} C_VEL
LIN {X 0,Y 319.606,Z 403.301,A -85,B 0,C 180,E1 -15272.498,E2 -15272.498} C_VEL
LIN {X 0,Y 319.604,Z 403.3,A -85,B 0,C 180,E1 -15275.304,E2 -15275.304} C_VEL
LIN {X 0,Y 319.605,Z 403.299,A -85,B 0,C 180,E1 -15279.4,E2 -15279.4} C_VEL
LIN {X 0,Y 319.66,Z 403.29,A -85,B 0,C 180,E1 -15282.073,E2 -15282.073} C_VEL
LIN {X 0,Y 319.733,Z 403.281,A -85,B 0,C 180,E1 -15286.008,E2 -15286.008} C_VEL
LIN {X 0,Y 319.759,Z 403.277,A -85,B 0,C 180,E1 -15289.873,E2 -15289.873} C_VEL
LIN {X 0,Y 319.935,Z 403.252,A -85,B 0,C 180,E1 -15292.426,E2 -15292.426} C_VEL
LIN {X 0,Y 319.749,Z 403.282,A -85,B 0,C 180,E1 -15294.956,E2 -15294.956} C_VEL
LIN {X 0,Y 319.993,Z 403.249,A -85,B 0,C 180,E1 -15297.483,E2 -15297.483} C_VEL
LIN {X 0,Y 320.17,Z 403.229,A -85,B 0,C 180,E1 -15300,E2 -15300} C_VEL
LIN {X 0,Y 319.991,Z 403.249,A -85,B 0,C 180,E1 -15302.518,E2 -15302.518} C_VEL
LIN {X 0,Y 319.932,Z 403.257,A -85,B 0,C 180,E1 -15306.668,E2 -15306.668} C_VEL
LIN {X 0,Y 319.76,Z 403.279,A -85,B 0,C 180,E1 -15310.127,E2 -15310.127} C_VEL
LIN {X 0,Y 319.732,Z 403.283,A -85,B 0,C 180,E1 -15314.724,E2 -15314.724} C_VEL
LIN {X 0,Y 319.691,Z 403.289,A -85,B 0,C 180,E1 -15319.038,E2 -15319.038} C_VEL
LIN {X 0,Y 319.571,Z 403.303,A -85,B 0,C 180,E1 -15323.319,E2 -15323.319} C_VEL
LIN {X 0,Y 319.635,Z 403.296,A -85,B 0,C 180,E1 -15326.088,E2 -15326.088} C_VEL
LIN {X 0,Y 319.581,Z 403.302,A -85,B 0,C 180,E1 -15328.935,E2 -15328.935} C_VEL
LIN {X 0,Y 319.533,Z 403.308,A -85,B 0,C 180,E1 -15331.862,E2 -15331.862} C_VEL
LIN {X 0,Y 319.582,Z 403.304,A -85,B 0,C 180,E1 -15335.543,E2 -15335.543} C_VEL
LIN {X 0,Y 319.575,Z 403.301,A -85,B 0,C 180,E1 -15338.008,E2 -15338.008} C_VEL
LIN {X 0,Y 319.527,Z 403.309,A -85,B 0,C 180,E1 -15341.597,E2 -15341.597} C_VEL
LIN {X 0,Y 319.548,Z 403.307,A -85,B 0,C 180,E1 -15345.268,E2 -15345.268} C_VEL
LIN {X 0,Y 319.986,Z 406.435,A -85,B 0,C 180,E1 -15348.784,E2 -15348.784} C_VEL
LIN {X 0,Y 319.994,Z 409.667,A -85,B 0,C 180,E1 -15352.051,E2 -15352.051} C_VEL
LIN {X 0,Y 319.82,Z 412.898,A -85,B 0,C 180,E1 -15355.156,E2 -15355.156} C_VEL
LIN {X 0,Y 319.386,Z 417.178,A -85,B 0,C 180,E1 -15359.114,E2 -15359.114} C_VEL
LIN {X 0,Y 319.12,Z 420.63,A -85,B 0,C 180,E1 -15362.194,E2 -15362.194} C_VEL
LIN {X 0,Y 321.084,Z 426.694,A -85,B 0,C 180,E1 -15362.581,E2 -15362.581} C_VEL
LIN {X 0,Y 325.344,Z 440.413,A -85,B 0,C 180,E1 -15363.591,E2 -15363.591} C_VEL
LIN {X 0,Y 328.402,Z 453.085,A -85,B 0,C 180,E1 -15364.659,E2 -15364.659} C_VEL
LIN {X 0,Y 330.478,Z 464.857,A -85,B 0,C 180,E1 -15365.786,E2 -15365.786} C_VEL
LIN {X 0,Y 330.351,Z 469.1,A -85,B 0,C 180,E1 -15366.177,E2 -15366.177} C_VEL
LIN {X 0,Y 328.815,Z 481.118,A -85,B 0,C 180,E1 -15367.373,E2 -15367.373} C_VEL
LIN {X 0,Y 326.841,Z 493.439,A -85,B 0,C 180,E1 -15368.889,E2 -15368.889} C_VEL
LIN {X 0,Y 325.056,Z 503.57,A -85,B 0,C 180,E1 -15370.42,E2 -15370.42} C_VEL
LIN {X 0,Y 323.245,Z 513.625,A -85,B 0,C 180,E1 -15372.279,E2 -15372.279} C_VEL
LIN {X 0,Y 321.798,Z 521.834,A -85,B 0,C 180,E1 -15374.121,E2 -15374.121} C_VEL
LIN {X 0,Y 320.658,Z 528.936,A -85,B 0,C 180,E1 -15376.049,E2 -15376.049} C_VEL
LIN {X 0,Y 319.567,Z 534.685,A -85,B 0,C 180,E1 -15377.941,E2 -15377.941} C_VEL
LIN {X 0,Y 318.874,Z 539.409,A -85,B 0,C 180,E1 -15379.845,E2 -15379.845} C_VEL
LIN {X 0,Y 318.232,Z 544.303,A -85,B 0,C 180,E1 -15382.386,E2 -15382.386} C_VEL
LIN {X 0,Y 317.914,Z 547.708,A -85,B 0,C 180,E1 -15384.927,E2 -15384.927} C_VEL
LIN {X 0,Y 317.761,Z 549.729,A -85,B 0,C 180,E1 -15387.465,E2 -15387.465} C_VEL
LIN {X 0,Y 317.704,Z 550.421,A -85,B 0,C 180,E1 -15390,E2 -15390} C_VEL
LIN {X 0,Y 317.76,Z 549.791,A -85,B 0,C 180,E1 -15392.535,E2 -15392.535} C_VEL
LIN {X 0,Y 317.913,Z 547.825,A -85,B 0,C 180,E1 -15395.073,E2 -15395.073} C_VEL
LIN {X 0,Y 318.226,Z 544.476,A -85,B 0,C 180,E1 -15397.615,E2 -15397.615} C_VEL
LIN {X 0,Y 318.844,Z 539.647,A -85,B 0,C 180,E1 -15400.157,E2 -15400.157} C_VEL
LIN {X 0,Y 319.538,Z 534.986,A -85,B 0,C 180,E1 -15402.061,E2 -15402.061} C_VEL
LIN {X 0,Y 320.832,Z 528.206,A -85,B 0,C 180,E1 -15404.267,E2 -15404.267} C_VEL
LIN {X 0,Y 321.987,Z 521.047,A -85,B 0,C 180,E1 -15406.18,E2 -15406.18} C_VEL
LIN {X 0,Y 323.492,Z 512.616,A -85,B 0,C 180,E1 -15408.035,E2 -15408.035} C_VEL
LIN {X 0,Y 325.336,Z 502.291,A -85,B 0,C 180,E1 -15409.891,E2 -15409.891} C_VEL
LIN {X 0,Y 327.35,Z 490.74,A -85,B 0,C 180,E1 -15411.572,E2 -15411.572} C_VEL
LIN {X 0,Y 329.158,Z 478.811,A -85,B 0,C 180,E1 -15412.979,E2 -15412.979} C_VEL
LIN {X 0,Y 330.642,Z 467.151,A -85,B 0,C 180,E1 -15414.093,E2 -15414.093} C_VEL
LIN {X 0,Y 329.31,Z 457.754,A -85,B 0,C 180,E1 -15415.026,E2 -15415.026} C_VEL
LIN {X 0,Y 326.463,Z 444.657,A -85,B 0,C 180,E1 -15416.183,E2 -15416.183} C_VEL
LIN {X 0,Y 322.515,Z 430.98,A -85,B 0,C 180,E1 -15417.234,E2 -15417.234} C_VEL
LIN {X 0,Y 319.123,Z 420.839,A -85,B 0,C 180,E1 -15417.902,E2 -15417.902} C_VEL
LIN {X 0,Y 319.472,Z 416.238,A -85,B 0,C 180,E1 -15421.869,E2 -15421.869} C_VEL
LIN {X 0,Y 319.876,Z 412.175,A -85,B 0,C 180,E1 -15425.617,E2 -15425.617} C_VEL
LIN {X 0,Y 319.994,Z 409.775,A -85,B 0,C 180,E1 -15427.949,E2 -15427.949} C_VEL
LIN {X 0,Y 320.013,Z 406.55,A -85,B 0,C 180,E1 -15431.212,E2 -15431.212} C_VEL
LIN {X 0,Y 319.556,Z 403.332,A -85,B 0,C 180,E1 -15434.731,E2 -15434.731} C_VEL
LIN {X 0,Y 319.528,Z 403.313,A -85,B 0,C 180,E1 -15438.403,E2 -15438.403} C_VEL
LIN {X 0,Y 319.56,Z 403.304,A -85,B 0,C 180,E1 -15441.99,E2 -15441.99} C_VEL
LIN {X 0,Y 319.563,Z 403.304,A -85,B 0,C 180,E1 -15445.124,E2 -15445.124} C_VEL
LIN {X 0,Y 319.573,Z 403.304,A -85,B 0,C 180,E1 -15449.058,E2 -15449.058} C_VEL
LIN {X 0,Y 319.611,Z 403.3,A -85,B 0,C 180,E1 -15452.498,E2 -15452.498} C_VEL
LIN {X 0,Y 319.598,Z 403.298,A -85,B 0,C 180,E1 -15453.075,E2 -15453.075} C_VEL
LIN {X 0,Y 318.937,Z 403.383,A -85,B 0,C 180,E1 -15454.127,E2 -15454.127} C_VEL
LIN {X 0,Y 316.074,Z 403.736,A -85,B 0,C 180,E1 -15455.838,E2 -15455.838} C_VEL
LIN {X 0,Y 313.651,Z 404.04,A -85,B 0,C 180,E1 -15457.225,E2 -15457.225} C_VEL
LIN {X 0,Y 312.626,Z 404.168,A -85,B 0,C 180,E1 -15458.3,E2 -15458.3} C_VEL
LIN {X 0,Y 312.551,Z 404.174,A -85,B 0,C 180,E1 -15458.664,E2 -15458.664} C_VEL
LIN {X 0,Y 312.641,Z 404.166,A -85,B 0,C 180,E1 -15461.656,E2 -15461.656} C_VEL
LIN {X 0,Y 312.696,Z 404.16,A -85,B 0,C 180,E1 -15465.686,E2 -15465.686} C_VEL
LIN {X 0,Y 312.705,Z 404.158,A -85,B 0,C 180,E1 -15469.642,E2 -15469.642} C_VEL
LIN {X 0,Y 312.875,Z 404.138,A -85,B 0,C 180,E1 -15472.254,E2 -15472.254} C_VEL
LIN {X 0,Y 312.721,Z 404.157,A -85,B 0,C 180,E1 -15474.842,E2 -15474.842} C_VEL
LIN {X 0,Y 312.991,Z 404.123,A -85,B 0,C 180,E1 -15478.713,E2 -15478.713} C_VEL
LIN {X 0,Y 312.994,Z 404.121,A -85,B 0,C 180,E1 -15481.287,E2 -15481.287} C_VEL
LIN {X 0,Y 312.721,Z 404.156,A -85,B 0,C 180,E1 -15485.157,E2 -15485.157} C_VEL
LIN {X 0,Y 312.875,Z 404.138,A -85,B 0,C 180,E1 -15487.746,E2 -15487.746} C_VEL
LIN {X 0,Y 312.672,Z 404.163,A -85,B 0,C 180,E1 -15491.671,E2 -15491.671} C_VEL
LIN {X 0,Y 312.702,Z 404.159,A -85,B 0,C 180,E1 -15494.888,E2 -15494.888} C_VEL
LIN {X 0,Y 312.634,Z 404.167,A -85,B 0,C 180,E1 -15499.237,E2 -15499.237} C_VEL
LIN {X 0,Y 312.548,Z 404.177,A -85,B 0,C 180,E1 -15502.789,E2 -15502.789} C_VEL
LIN {X 0,Y 312.604,Z 404.172,A -85,B 0,C 180,E1 -15505.935,E2 -15505.935} C_VEL
LIN {X 0,Y 312.54,Z 404.176,A -85,B 0,C 180,E1 -15509.65,E2 -15509.65} C_VEL
LIN {X 0,Y 312.521,Z 404.184,A -85,B 0,C 180,E1 -15513.689,E2 -15513.689} C_VEL
LIN {X 0,Y 312.555,Z 404.183,A -85,B 0,C 180,E1 -15517.381,E2 -15517.381} C_VEL
LIN {X 0,Y 312.514,Z 404.186,A -85,B 0,C 180,E1 -15521.398,E2 -15521.398} C_VEL
LIN {X 0,Y 312.547,Z 404.265,A -85,B 0,C 180,E1 -15522.094,E2 -15522.094} C_VEL
LIN {X 0,Y 313.122,Z 407.883,A -85,B 0,C 180,E1 -15525.909,E2 -15525.909} C_VEL
LIN {X 0,Y 313.489,Z 411.524,A -85,B 0,C 180,E1 -15529.447,E2 -15529.447} C_VEL
LIN {X 0,Y 313.481,Z 414,A -85,B 0,C 180,E1 -15531.691,E2 -15531.691} C_VEL
LIN {X 0,Y 313.228,Z 416.979,A -85,B 0,C 180,E1 -15534.312,E2 -15534.312} C_VEL
LIN {X 0,Y 312.741,Z 420.63,A -85,B 0,C 180,E1 -15537.361,E2 -15537.361} C_VEL
LIN {X 0,Y 312.221,Z 425.715,A -85,B 0,C 180,E1 -15541.455,E2 -15541.455} C_VEL
LIN {X 0,Y 314.147,Z 431.758,A -85,B 0,C 180,E1 -15541.837,E2 -15541.837} C_VEL
LIN {X 0,Y 318.343,Z 446.033,A -85,B 0,C 180,E1 -15542.896,E2 -15542.896} C_VEL
LIN {X 0,Y 321.361,Z 459.649,A -85,B 0,C 180,E1 -15544.062,E2 -15544.062} C_VEL
LIN {X 0,Y 323.214,Z 471.552,A -85,B 0,C 180,E1 -15545.228,E2 -15545.228} C_VEL
LIN {X 0,Y 323.612,Z 475.368,A -85,B 0,C 180,E1 -15545.63,E2 -15545.63} C_VEL
LIN {X 0,Y 321.88,Z 487.477,A -85,B 0,C 180,E1 -15546.857,E2 -15546.857} C_VEL
LIN {X 0,Y 319.797,Z 499.695,A -85,B 0,C 180,E1 -15548.401,E2 -15548.401} C_VEL
LIN {X 0,Y 317.991,Z 509.783,A -85,B 0,C 180,E1 -15549.966,E2 -15549.966} C_VEL
LIN {X 0,Y 316.1,Z 519.812,A -85,B 0,C 180,E1 -15551.864,E2 -15551.864} C_VEL
LIN {X 0,Y 314.392,Z 528.958,A -85,B 0,C 180,E1 -15553.994,E2 -15553.994} C_VEL
LIN {X 0,Y 313.067,Z 537.117,A -85,B 0,C 180,E1 -15556.366,E2 -15556.366} C_VEL
LIN {X 0,Y 312.048,Z 542.519,A -85,B 0,C 180,E1 -15558.305,E2 -15558.305} C_VEL
LIN {X 0,Y 311.292,Z 548.204,A -85,B 0,C 180,E1 -15560.907,E2 -15560.907} C_VEL
LIN {X 0,Y 310.834,Z 552.328,A -85,B 0,C 180,E1 -15563.509,E2 -15563.509} C_VEL
LIN {X 0,Y 310.685,Z 555.021,A -85,B 0,C 180,E1 -15566.109,E2 -15566.109} C_VEL
LIN {X 0,Y 310.606,Z 556.353,A -85,B 0,C 180,E1 -15568.703,E2 -15568.703} C_VEL
LIN {X 0,Y 310.605,Z 556.349,A -85,B 0,C 180,E1 -15571.296,E2 -15571.296} C_VEL
LIN {X 0,Y 310.686,Z 555.009,A -85,B 0,C 180,E1 -15573.891,E2 -15573.891} C_VEL
LIN {X 0,Y 310.838,Z 552.308,A -85,B 0,C 180,E1 -15576.491,E2 -15576.491} C_VEL
LIN {X 0,Y 311.275,Z 548.17,A -85,B 0,C 180,E1 -15579.093,E2 -15579.093} C_VEL
LIN {X 0,Y 312.046,Z 542.473,A -85,B 0,C 180,E1 -15581.695,E2 -15581.695} C_VEL
LIN {X 0,Y 313.266,Z 536.052,A -85,B 0,C 180,E1 -15583.956,E2 -15583.956} C_VEL
LIN {X 0,Y 314.612,Z 527.93,A -85,B 0,C 180,E1 -15586.253,E2 -15586.253} C_VEL
LIN {X 0,Y 316.095,Z 519.728,A -85,B 0,C 180,E1 -15588.136,E2 -15588.136} C_VEL
LIN {X 0,Y 318.005,Z 509.681,A -85,B 0,C 180,E1 -15590.033,E2 -15590.033} C_VEL
LIN {X 0,Y 320.017,Z 498.469,A -85,B 0,C 180,E1 -15591.752,E2 -15591.752} C_VEL
LIN {X 0,Y 322.016,Z 486.313,A -85,B 0,C 180,E1 -15593.251,E2 -15593.251} C_VEL
LIN {X 0,Y 323.544,Z 475.161,A -85,B 0,C 180,E1 -15594.376,E2 -15594.376} C_VEL
LIN {X 0,Y 322.218,Z 464.504,A -85,B 0,C 180,E1 -15595.46,E2 -15595.46} C_VEL
LIN {X 0,Y 319.782,Z 452.062,A -85,B 0,C 180,E1 -15596.588,E2 -15596.588} C_VEL
LIN {X 0,Y 316.248,Z 438.677,A -85,B 0,C 180,E1 -15597.652,E2 -15597.652} C_VEL
LIN {X 0,Y 312.195,Z 425.638,A -85,B 0,C 180,E1 -15598.555,E2 -15598.555} C_VEL
LIN {X 0,Y 312.555,Z 422.238,A -85,B 0,C 180,E1 -15601.301,E2 -15601.301} C_VEL
LIN {X 0,Y 312.984,Z 418.78,A -85,B 0,C 180,E1 -15604.151,E2 -15604.151} C_VEL
LIN {X 0,Y 313.377,Z 415.142,A -85,B 0,C 180,E1 -15607.266,E2 -15607.266} C_VEL
LIN {X 0,Y 313.485,Z 411.485,A -85,B 0,C 180,E1 -15610.553,E2 -15610.553} C_VEL
LIN {X 0,Y 313.1,Z 407.863,A -85,B 0,C 180,E1 -15614.094,E2 -15614.094} C_VEL
LIN {X 0,Y 312.544,Z 404.183,A -85,B 0,C 180,E1 -15617.96,E2 -15617.96} C_VEL
LIN {X 0,Y 312.558,Z 404.178,A -85,B 0,C 180,E1 -15621.905,E2 -15621.905} C_VEL
LIN {X 0,Y 312.507,Z 404.186,A -85,B 0,C 180,E1 -15625.79,E2 -15625.79} C_VEL
LIN {X 0,Y 312.521,Z 404.184,A -85,B 0,C 180,E1 -15628.854,E2 -15628.854} C_VEL
LIN {X 0,Y 312.571,Z 404.176,A -85,B 0,C 180,E1 -15631.824,E2 -15631.824} C_VEL
LIN {X 0,Y 312.585,Z 404.174,A -85,B 0,C 180,E1 -15634.711,E2 -15634.711} C_VEL
LIN {X 0,Y 312.539,Z 404.181,A -85,B 0,C 180,E1 -15638.913,E2 -15638.913} C_VEL
LIN {X 0,Y 312.64,Z 404.166,A -85,B 0,C 180,E1 -15641.657,E2 -15641.657} C_VEL
LIN {X 0,Y 312.695,Z 404.157,A -85,B 0,C 180,E1 -15645.686,E2 -15645.686} C_VEL
LIN {X 0,Y 312.703,Z 404.155,A -85,B 0,C 180,E1 -15649.642,E2 -15649.642} C_VEL
LIN {X 0,Y 312.873,Z 404.133,A -85,B 0,C 180,E1 -15652.254,E2 -15652.254} C_VEL
LIN {X 0,Y 312.72,Z 404.157,A -85,B 0,C 180,E1 -15654.843,E2 -15654.843} C_VEL
LIN {X 0,Y 312.992,Z 404.123,A -85,B 0,C 180,E1 -15658.713,E2 -15658.713} C_VEL
LIN {X 0,Y 313.122,Z 404.107,A -85,B 0,C 180,E1 -15660,E2 -15660} C_VEL
LIN {X 0,Y 312.938,Z 404.128,A -85,B 0,C 180,E1 -15662.574,E2 -15662.574} C_VEL
LIN {X 0,Y 312.895,Z 404.134,A -85,B 0,C 180,E1 -15666.651,E2 -15666.651} C_VEL
LIN {X 0,Y 312.789,Z 404.147,A -85,B 0,C 180,E1 -15669.049,E2 -15669.049} C_VEL
LIN {X 0,Y 312.636,Z 404.164,A -85,B 0,C 180,E1 -15672.991,E2 -15672.991} C_VEL
LIN {X 0,Y 312.64,Z 404.166,A -85,B 0,C 180,E1 -15675.65,E2 -15675.65} C_VEL
LIN {X 0,Y 312.633,Z 404.169,A -85,B 0,C 180,E1 -15679.237,E2 -15679.237} C_VEL
LIN {X 0,Y 312.547,Z 404.179,A -85,B 0,C 180,E1 -15682.789,E2 -15682.789} C_VEL
LIN {X 0,Y 312.604,Z 404.172,A -85,B 0,C 180,E1 -15685.936,E2 -15685.936} C_VEL
LIN {X 0,Y 312.539,Z 404.179,A -85,B 0,C 180,E1 -15689.651,E2 -15689.651} C_VEL
LIN {X 0,Y 312.521,Z 404.182,A -85,B 0,C 180,E1 -15693.689,E2 -15693.689} C_VEL
LIN {X 0,Y 312.539,Z 404.181,A -85,B 0,C 180,E1 -15697.383,E2 -15697.383} C_VEL
LIN {X 0,Y 312.491,Z 404.187,A -85,B 0,C 180,E1 -15700.709,E2 -15700.709} C_VEL
LIN {X 0,Y 312.476,Z 404.185,A -85,B 0,C 180,E1 -15704.206,E2 -15704.206} C_VEL
LIN {X 0,Y 312.624,Z 405.056,A -85,B 0,C 180,E1 -15706.004,E2 -15706.004} C_VEL
LIN {X 0,Y 312.976,Z 408.12,A -85,B 0,C 180,E1 -15709.367,E2 -15709.367} C_VEL
LIN {X 0,Y 312.923,Z 411.333,A -85,B 0,C 180,E1 -15712.671,E2 -15712.671} C_VEL
LIN {X 0,Y 312.695,Z 414.58,A -85,B 0,C 180,E1 -15715.814,E2 -15715.814} C_VEL
LIN {X 0,Y 312.358,Z 417.786,A -85,B 0,C 180,E1 -15718.836,E2 -15718.836} C_VEL
LIN {X 0,Y 312.124,Z 420.912,A -85,B 0,C 180,E1 -15721.531,E2 -15721.531} C_VEL
LIN {X 0,Y 316.83,Z 435.002,A -85,B 0,C 180,E1 -15722.535,E2 -15722.535} C_VEL
LIN {X 0,Y 320.328,Z 447.777,A -85,B 0,C 180,E1 -15723.592,E2 -15723.592} C_VEL
LIN {X 0,Y 322.765,Z 459.348,A -85,B 0,C 180,E1 -15724.674,E2 -15724.674} C_VEL
LIN {X 0,Y 323.999,Z 467.73,A -85,B 0,C 180,E1 -15725.541,E2 -15725.541} C_VEL
LIN {X 0,Y 322.463,Z 480.13,A -85,B 0,C 180,E1 -15726.775,E2 -15726.775} C_VEL
LIN {X 0,Y 320.405,Z 492.387,A -85,B 0,C 180,E1 -15728.275,E2 -15728.275} C_VEL
LIN {X 0,Y 318.364,Z 503.642,A -85,B 0,C 180,E1 -15729.991,E2 -15729.991} C_VEL
LIN {X 0,Y 316.461,Z 513.697,A -85,B 0,C 180,E1 -15731.886,E2 -15731.886} C_VEL
LIN {X 0,Y 314.85,Z 522.392,A -85,B 0,C 180,E1 -15733.893,E2 -15733.893} C_VEL
LIN {X 0,Y 313.539,Z 530.014,A -85,B 0,C 180,E1 -15736.057,E2 -15736.057} C_VEL
LIN {X 0,Y 312.333,Z 536.431,A -85,B 0,C 180,E1 -15738.316,E2 -15738.316} C_VEL
LIN {X 0,Y 311.451,Z 542.12,A -85,B 0,C 180,E1 -15740.912,E2 -15740.912} C_VEL
LIN {X 0,Y 310.988,Z 546.253,A -85,B 0,C 180,E1 -15743.512,E2 -15743.512} C_VEL
LIN {X 0,Y 310.753,Z 548.956,A -85,B 0,C 180,E1 -15746.11,E2 -15746.11} C_VEL
LIN {X 0,Y 310.618,Z 550.309,A -85,B 0,C 180,E1 -15748.704,E2 -15748.704} C_VEL
LIN {X 0,Y 310.618,Z 550.34,A -85,B 0,C 180,E1 -15751.297,E2 -15751.297} C_VEL
LIN {X 0,Y 310.752,Z 549.045,A -85,B 0,C 180,E1 -15753.891,E2 -15753.891} C_VEL
LIN {X 0,Y 310.988,Z 546.396,A -85,B 0,C 180,E1 -15756.488,E2 -15756.488} C_VEL
LIN {X 0,Y 311.441,Z 542.324,A -85,B 0,C 180,E1 -15759.089,E2 -15759.089} C_VEL
LIN {X 0,Y 312.305,Z 536.698,A -85,B 0,C 180,E1 -15761.685,E2 -15761.685} C_VEL
LIN {X 0,Y 313.501,Z 530.344,A -85,B 0,C 180,E1 -15763.945,E2 -15763.945} C_VEL
LIN {X 0,Y 314.859,Z 522.772,A -85,B 0,C 180,E1 -15766.113,E2 -15766.113} C_VEL
LIN {X 0,Y 316.435,Z 514.18,A -85,B 0,C 180,E1 -15768.116,E2 -15768.116} C_VEL
LIN {X 0,Y 318.291,Z 504.222,A -85,B 0,C 180,E1 -15770.014,E2 -15770.014} C_VEL
LIN {X 0,Y 320.328,Z 493.133,A -85,B 0,C 180,E1 -15771.73,E2 -15771.73} C_VEL
LIN {X 0,Y 322.152,Z 482.092,A -85,B 0,C 180,E1 -15773.122,E2 -15773.122} C_VEL
LIN {X 0,Y 323.85,Z 470.103,A -85,B 0,C 180,E1 -15774.351,E2 -15774.351} C_VEL
LIN {X 0,Y 323.866,Z 466.091,A -85,B 0,C 180,E1 -15774.74,E2 -15774.74} C_VEL
LIN {X 0,Y 321.67,Z 453.459,A -85,B 0,C 180,E1 -15776.001,E2 -15776.001} C_VEL
LIN {X 0,Y 318.334,Z 440.085,A -85,B 0,C 180,E1 -15777.176,E2 -15777.176} C_VEL
LIN {X 0,Y 314.013,Z 426.451,A -85,B 0,C 180,E1 -15778.218,E2 -15778.218} C_VEL
LIN {X 0,Y 312.125,Z 421.054,A -85,B 0,C 180,E1 -15778.58,E2 -15778.58} C_VEL
LIN {X 0,Y 312.095,Z 420.644,A -85,B 0,C 180,E1 -15778.668,E2 -15778.668} C_VEL
LIN {X 0,Y 312.51,Z 416.279,A -85,B 0,C 180,E1 -15782.666,E2 -15782.666} C_VEL
LIN {X 0,Y 312.867,Z 412.762,A -85,B 0,C 180,E1 -15786.033,E2 -15786.033} C_VEL
LIN {X 0,Y 312.998,Z 409.835,A -85,B 0,C 180,E1 -15788.955,E2 -15788.955} C_VEL
LIN {X 0,Y 312.867,Z 406.813,A -85,B 0,C 180,E1 -15792.159,E2 -15792.159} C_VEL
LIN {X 0,Y 312.628,Z 405.002,A -85,B 0,C 180,E1 -15794.178,E2 -15794.178} C_VEL
LIN {X 0,Y 312.485,Z 404.191,A -85,B 0,C 180,E1 -15796.03,E2 -15796.03} C_VEL
LIN {X 0,Y 312.506,Z 404.186,A -85,B 0,C 180,E1 -15799.875,E2 -15799.875} C_VEL
LIN {X 0,Y 312.538,Z 404.179,A -85,B 0,C 180,E1 -15804.05,E2 -15804.05} C_VEL
LIN {X 0,Y 312.507,Z 404.185,A -85,B 0,C 180,E1 -15807.334,E2 -15807.334} C_VEL
LIN {X 0,Y 312.554,Z 404.178,A -85,B 0,C 180,E1 -15811.276,E2 -15811.276} C_VEL
LIN {X 0,Y 312.588,Z 404.173,A -85,B 0,C 180,E1 -15814.711,E2 -15814.711} C_VEL
LIN {X 0,Y 312.551,Z 404.174,A -85,B 0,C 180,E1 -15818.664,E2 -15818.664} C_VEL
LIN {X 0,Y 311.907,Z 404.257,A -85,B 0,C 180,E1 -15819.739,E2 -15819.739} C_VEL
LIN {X 0,Y 309.074,Z 404.613,A -85,B 0,C 180,E1 -15821.491,E2 -15821.491} C_VEL
LIN {X 0,Y 306.678,Z 404.91,A -85,B 0,C 180,E1 -15822.912,E2 -15822.912} C_VEL
LIN {X 0,Y 305.672,Z 405.034,A -85,B 0,C 180,E1 -15824.012,E2 -15824.012} C_VEL
LIN {X 0,Y 305.604,Z 405.041,A -85,B 0,C 180,E1 -15824.384,E2 -15824.384} C_VEL
LIN {X 0,Y 305.606,Z 405.042,A -85,B 0,C 180,E1 -15828.055,E2 -15828.055} C_VEL
LIN {X 0,Y 305.816,Z 405.018,A -85,B 0,C 180,E1 -15832.074,E2 -15832.074} C_VEL
LIN {X 0,Y 305.692,Z 405.032,A -85,B 0,C 180,E1 -15834.723,E2 -15834.723} C_VEL
LIN {X 0,Y 305.958,Z 404.999,A -85,B 0,C 180,E1 -15838.684,E2 -15838.684} C_VEL
LIN {X 0,Y 305.96,Z 404.997,A -85,B 0,C 180,E1 -15841.316,E2 -15841.316} C_VEL
LIN {X 0,Y 305.855,Z 405.014,A -85,B 0,C 180,E1 -15846.597,E2 -15846.597} C_VEL
LIN {X 0,Y 305.738,Z 405.026,A -85,B 0,C 180,E1 -15849.26,E2 -15849.26} C_VEL
LIN {X 0,Y 305.592,Z 405.046,A -85,B 0,C 180,E1 -15853.296,E2 -15853.296} C_VEL
LIN {X 0,Y 305.596,Z 405.045,A -85,B 0,C 180,E1 -15856.02,E2 -15856.02} C_VEL
LIN {X 0,Y 305.58,Z 405.046,A -85,B 0,C 180,E1 -15859.445,E2 -15859.445} C_VEL
LIN {X 0,Y 305.492,Z 405.054,A -85,B 0,C 180,E1 -15863.041,E2 -15863.041} C_VEL
LIN {X 0,Y 305.533,Z 405.051,A -85,B 0,C 180,E1 -15866.221,E2 -15866.221} C_VEL
LIN {X 0,Y 305.49,Z 405.058,A -85,B 0,C 180,E1 -15869.047,E2 -15869.047} C_VEL
LIN {X 0,Y 305.444,Z 405.063,A -85,B 0,C 180,E1 -15871.952,E2 -15871.952} C_VEL
LIN {X 0,Y 305.465,Z 405.062,A -85,B 0,C 180,E1 -15875.113,E2 -15875.113} C_VEL
LIN {X 0,Y 305.494,Z 405.062,A -85,B 0,C 180,E1 -15878.539,E2 -15878.539} C_VEL
LIN {X 0,Y 305.537,Z 405.316,A -85,B 0,C 180,E1 -15881.841,E2 -15881.841} C_VEL
LIN {X 0,Y 306.027,Z 408.598,A -85,B 0,C 180,E1 -15885.392,E2 -15885.392} C_VEL
LIN {X 0,Y 306.378,Z 411.471,A -85,B 0,C 180,E1 -15888.3,E2 -15888.3} C_VEL
LIN {X 0,Y 306.503,Z 414.536,A -85,B 0,C 180,E1 -15891.225,E2 -15891.225} C_VEL
LIN {X 0,Y 306.289,Z 416.998,A -85,B 0,C 180,E1 -15893.427,E2 -15893.427} C_VEL
LIN {X 0,Y 305.819,Z 420.551,A -85,B 0,C 180,E1 -15896.527,E2 -15896.527} C_VEL
LIN {X 0,Y 305.25,Z 425.785,A -85,B 0,C 180,E1 -15900.745,E2 -15900.745} C_VEL
LIN {X 0,Y 307.107,Z 431.479,A -85,B 0,C 180,E1 -15901.123,E2 -15901.123} C_VEL
LIN {X 0,Y 311.153,Z 444.705,A -85,B 0,C 180,E1 -15902.141,E2 -15902.141} C_VEL
LIN {X 0,Y 314.431,Z 458.839,A -85,B 0,C 180,E1 -15903.388,E2 -15903.388} C_VEL
LIN {X 0,Y 316.343,Z 470.634,A -85,B 0,C 180,E1 -15904.568,E2 -15904.568} C_VEL
LIN {X 0,Y 316.982,Z 476.489,A -85,B 0,C 180,E1 -15905.21,E2 -15905.21} C_VEL
LIN {X 0,Y 315.136,Z 488.729,A -85,B 0,C 180,E1 -15906.507,E2 -15906.507} C_VEL
LIN {X 0,Y 312.975,Z 500.699,A -85,B 0,C 180,E1 -15908.079,E2 -15908.079} C_VEL
LIN {X 0,Y 310.94,Z 511.5,A -85,B 0,C 180,E1 -15909.837,E2 -15909.837} C_VEL
LIN {X 0,Y 309.023,Z 521.233,A -85,B 0,C 180,E1 -15911.777,E2 -15911.777} C_VEL
LIN {X 0,Y 307.449,Z 529.373,A -85,B 0,C 180,E1 -15913.756,E2 -15913.756} C_VEL
LIN {X 0,Y 306.143,Z 537.049,A -85,B 0,C 180,E1 -15916.052,E2 -15916.052} C_VEL
LIN {X 0,Y 305.055,Z 542.45,A -85,B 0,C 180,E1 -15918.033,E2 -15918.033} C_VEL
LIN {X 0,Y 304.247,Z 548.135,A -85,B 0,C 180,E1 -15920.694,E2 -15920.694} C_VEL
LIN {X 0,Y 303.748,Z 552.259,A -85,B 0,C 180,E1 -15923.357,E2 -15923.357} C_VEL
LIN {X 0,Y 303.583,Z 554.953,A -85,B 0,C 180,E1 -15926.017,E2 -15926.017} C_VEL
LIN {X 0,Y 303.525,Z 556.285,A -85,B 0,C 180,E1 -15928.673,E2 -15928.673} C_VEL
LIN {X 0,Y 303.525,Z 556.28,A -85,B 0,C 180,E1 -15931.327,E2 -15931.327} C_VEL
LIN {X 0,Y 303.584,Z 554.94,A -85,B 0,C 180,E1 -15933.982,E2 -15933.982} C_VEL
LIN {X 0,Y 303.752,Z 552.239,A -85,B 0,C 180,E1 -15936.643,E2 -15936.643} C_VEL
LIN {X 0,Y 304.23,Z 548.1,A -85,B 0,C 180,E1 -15939.306,E2 -15939.306} C_VEL
LIN {X 0,Y 305.053,Z 542.402,A -85,B 0,C 180,E1 -15941.967,E2 -15941.967} C_VEL
LIN {X 0,Y 306.33,Z 535.981,A -85,B 0,C 180,E1 -15944.278,E2 -15944.278} C_VEL
LIN {X 0,Y 307.701,Z 528.164,A -85,B 0,C 180,E1 -15946.544,E2 -15946.544} C_VEL
LIN {X 0,Y 309.331,Z 519.656,A -85,B 0,C 180,E1 -15948.547,E2 -15948.547} C_VEL
LIN {X 0,Y 311.328,Z 509.609,A -85,B 0,C 180,E1 -15950.481,E2 -15950.481} C_VEL
LIN {X 0,Y 313.428,Z 498.397,A -85,B 0,C 180,E1 -15952.234,E2 -15952.234} C_VEL
LIN {X 0,Y 315.344,Z 487.242,A -85,B 0,C 180,E1 -15953.651,E2 -15953.651} C_VEL
LIN {X 0,Y 316.906,Z 476.304,A -85,B 0,C 180,E1 -15954.795,E2 -15954.795} C_VEL
LIN {X 0,Y 315.392,Z 464.281,A -85,B 0,C 180,E1 -15956.065,E2 -15956.065} C_VEL
LIN {X 0,Y 312.961,Z 452.097,A -85,B 0,C 180,E1 -15957.206,E2 -15957.206} C_VEL
LIN {X 0,Y 309.219,Z 437.956,A -85,B 0,C 180,E1 -15958.368,E2 -15958.368} C_VEL
LIN {X 0,Y 305.384,Z 426.671,A -85,B 0,C 180,E1 -15959.187,E2 -15959.187} C_VEL
LIN {X 0,Y 305.234,Z 425.579,A -85,B 0,C 180,E1 -15959.266,E2 -15959.266} C_VEL
LIN {X 0,Y 305.818,Z 420.527,A -85,B 0,C 180,E1 -15963.473,E2 -15963.473} C_VEL
LIN {X 0,Y 306.29,Z 416.892,A -85,B 0,C 180,E1 -15966.626,E2 -15966.626} C_VEL
LIN {X 0,Y 306.48,Z 413.25,A -85,B 0,C 180,E1 -15969.947,E2 -15969.947} C_VEL
LIN {X 0,Y 306.18,Z 409.61,A -85,B 0,C 180,E1 -15973.52,E2 -15973.52} C_VEL
LIN {X 0,Y 305.679,Z 405.984,A -85,B 0,C 180,E1 -15977.369,E2 -15977.369} C_VEL
LIN {X 0,Y 305.531,Z 405.28,A -85,B 0,C 180,E1 -15978.158,E2 -15978.158} C_VEL
LIN {X 0,Y 305.519,Z 405.055,A -85,B 0,C 180,E1 -15981.604,E2 -15981.604} C_VEL
LIN {X 0,Y 305.464,Z 405.062,A -85,B 0,C 180,E1 -15984.887,E2 -15984.887} C_VEL
LIN {X 0,Y 305.45,Z 405.064,A -85,B 0,C 180,E1 -15988.356,E2 -15988.356} C_VEL
LIN {X 0,Y 305.514,Z 405.056,A -85,B 0,C 180,E1 -15991.113,E2 -15991.113} C_VEL
LIN {X 0,Y 305.571,Z 405.048,A -85,B 0,C 180,E1 -15994.088,E2 -15994.088} C_VEL
LIN {X 0,Y 305.483,Z 405.058,A -85,B 0,C 180,E1 -15998.402,E2 -15998.402} C_VEL
LIN {X 0,Y 305.591,Z 405.044,A -85,B 0,C 180,E1 -16001.218,E2 -16001.218} C_VEL
LIN {X 0,Y 305.65,Z 405.034,A -85,B 0,C 180,E1 -16005.349,E2 -16005.349} C_VEL
LIN {X 0,Y 305.64,Z 405.035,A -85,B 0,C 180,E1 -16009.4,E2 -16009.4} C_VEL
LIN {X 0,Y 305.814,Z 405.013,A -85,B 0,C 180,E1 -16012.074,E2 -16012.074} C_VEL
LIN {X 0,Y 305.691,Z 405.032,A -85,B 0,C 180,E1 -16014.724,E2 -16014.724} C_VEL
LIN {X 0,Y 305.959,Z 405,A -85,B 0,C 180,E1 -16018.684,E2 -16018.684} C_VEL
LIN {X 0,Y 305.959,Z 405,A -85,B 0,C 180,E1 -16021.316,E2 -16021.316} C_VEL
LIN {X 0,Y 305.851,Z 405.012,A -85,B 0,C 180,E1 -16026.63,E2 -16026.63} C_VEL
LIN {X 0,Y 305.737,Z 405.026,A -85,B 0,C 180,E1 -16029.26,E2 -16029.26} C_VEL
LIN {X 0,Y 305.59,Z 405.04,A -85,B 0,C 180,E1 -16033.296,E2 -16033.296} C_VEL
LIN {X 0,Y 305.595,Z 405.045,A -85,B 0,C 180,E1 -16036.02,E2 -16036.02} C_VEL
LIN {X 0,Y 305.579,Z 405.047,A -85,B 0,C 180,E1 -16039.446,E2 -16039.446} C_VEL
LIN {X 0,Y 305.492,Z 405.058,A -85,B 0,C 180,E1 -16043.042,E2 -16043.042} C_VEL
LIN {X 0,Y 305.548,Z 405.051,A -85,B 0,C 180,E1 -16046.227,E2 -16046.227} C_VEL
LIN {X 0,Y 305.489,Z 405.058,A -85,B 0,C 180,E1 -16049.048,E2 -16049.048} C_VEL
LIN {X 0,Y 305.444,Z 405.063,A -85,B 0,C 180,E1 -16051.952,E2 -16051.952} C_VEL
LIN {X 0,Y 305.464,Z 405.061,A -85,B 0,C 180,E1 -16055.113,E2 -16055.113} C_VEL
LIN {X 0,Y 305.468,Z 405.059,A -85,B 0,C 180,E1 -16058.533,E2 -16058.533} C_VEL
LIN {X 0,Y 305.46,Z 405.062,A -85,B 0,C 180,E1 -16062.587,E2 -16062.587} C_VEL
LIN {X 0,Y 305.437,Z 405.063,A -85,B 0,C 180,E1 -16064.496,E2 -16064.496} C_VEL
LIN {X 0,Y 305.865,Z 408.19,A -85,B 0,C 180,E1 -16068.214,E2 -16068.214} C_VEL
LIN {X 0,Y 305.96,Z 411.1,A -85,B 0,C 180,E1 -16071.352,E2 -16071.352} C_VEL
LIN {X 0,Y 305.721,Z 414.625,A -85,B 0,C 180,E1 -16074.921,E2 -16074.921} C_VEL
LIN {X 0,Y 305.373,Z 418.217,A -85,B 0,C 180,E1 -16078.38,E2 -16078.38} C_VEL
LIN {X 0,Y 305.109,Z 420.849,A -85,B 0,C 180,E1 -16080.809,E2 -16080.809} C_VEL
LIN {X 0,Y 306.082,Z 423.915,A -85,B 0,C 180,E1 -16081.007,E2 -16081.007} C_VEL
LIN {X 0,Y 310.266,Z 436.138,A -85,B 0,C 180,E1 -16081.956,E2 -16081.956} C_VEL
LIN {X 0,Y 313.86,Z 449.254,A -85,B 0,C 180,E1 -16083.101,E2 -16083.101} C_VEL
LIN {X 0,Y 316.417,Z 461.985,A -85,B 0,C 180,E1 -16084.357,E2 -16084.357} C_VEL
LIN {X 0,Y 317.394,Z 469.049,A -85,B 0,C 180,E1 -16085.12,E2 -16085.12} C_VEL
LIN {X 0,Y 315.766,Z 481.265,A -85,B 0,C 180,E1 -16086.383,E2 -16086.383} C_VEL
LIN {X 0,Y 313.605,Z 493.585,A -85,B 0,C 180,E1 -16087.953,E2 -16087.953} C_VEL
LIN {X 0,Y 311.683,Z 503.714,A -85,B 0,C 180,E1 -16089.543,E2 -16089.543} C_VEL
LIN {X 0,Y 309.681,Z 513.768,A -85,B 0,C 180,E1 -16091.475,E2 -16091.475} C_VEL
LIN {X 0,Y 307.902,Z 522.963,A -85,B 0,C 180,E1 -16093.658,E2 -16093.658} C_VEL
LIN {X 0,Y 306.629,Z 530.085,A -85,B 0,C 180,E1 -16095.736,E2 -16095.736} C_VEL
LIN {X 0,Y 305.335,Z 536.502,A -85,B 0,C 180,E1 -16098.044,E2 -16098.044} C_VEL
LIN {X 0,Y 304.428,Z 542.19,A -85,B 0,C 180,E1 -16100.7,E2 -16100.7} C_VEL
LIN {X 0,Y 303.92,Z 546.323,A -85,B 0,C 180,E1 -16103.361,E2 -16103.361} C_VEL
LIN {X 0,Y 303.671,Z 549.025,A -85,B 0,C 180,E1 -16106.019,E2 -16106.019} C_VEL
LIN {X 0,Y 303.538,Z 550.378,A -85,B 0,C 180,E1 -16108.673,E2 -16108.673} C_VEL
LIN {X 0,Y 303.538,Z 550.409,A -85,B 0,C 180,E1 -16111.327,E2 -16111.327} C_VEL
LIN {X 0,Y 303.67,Z 549.114,A -85,B 0,C 180,E1 -16113.981,E2 -16113.981} C_VEL
LIN {X 0,Y 303.92,Z 546.464,A -85,B 0,C 180,E1 -16116.64,E2 -16116.64} C_VEL
LIN {X 0,Y 304.417,Z 542.392,A -85,B 0,C 180,E1 -16119.3,E2 -16119.3} C_VEL
LIN {X 0,Y 305.307,Z 536.766,A -85,B 0,C 180,E1 -16121.957,E2 -16121.957} C_VEL
LIN {X 0,Y 306.594,Z 530.411,A -85,B 0,C 180,E1 -16124.266,E2 -16124.266} C_VEL
LIN {X 0,Y 308.072,Z 522.27,A -85,B 0,C 180,E1 -16126.636,E2 -16126.636} C_VEL
LIN {X 0,Y 309.656,Z 514.247,A -85,B 0,C 180,E1 -16128.527,E2 -16128.527} C_VEL
LIN {X 0,Y 311.61,Z 504.288,A -85,B 0,C 180,E1 -16130.462,E2 -16130.462} C_VEL
LIN {X 0,Y 313.741,Z 493.198,A -85,B 0,C 180,E1 -16132.211,E2 -16132.211} C_VEL
LIN {X 0,Y 315.626,Z 482.157,A -85,B 0,C 180,E1 -16133.629,E2 -16133.629} C_VEL
LIN {X 0,Y 317.39,Z 470.166,A -85,B 0,C 180,E1 -16134.88,E2 -16134.88} C_VEL
LIN {X 0,Y 316.96,Z 465.263,A -85,B 0,C 180,E1 -16135.406,E2 -16135.406} C_VEL
LIN {X 0,Y 314.648,Z 452.716,A -85,B 0,C 180,E1 -16136.69,E2 -16136.69} C_VEL
LIN {X 0,Y 311.213,Z 439.288,A -85,B 0,C 180,E1 -16137.903,E2 -16137.903} C_VEL
LIN {X 0,Y 307.294,Z 427.127,A -85,B 0,C 180,E1 -16138.867,E2 -16138.867} C_VEL
LIN {X 0,Y 305.144,Z 421.222,A -85,B 0,C 180,E1 -16139.293,E2 -16139.293} C_VEL
LIN {X 0,Y 305.073,Z 420.747,A -85,B 0,C 180,E1 -16139.349,E2 -16139.349} C_VEL
LIN {X 0,Y 305.387,Z 417.965,A -85,B 0,C 180,E1 -16141.959,E2 -16141.959} C_VEL
LIN {X 0,Y 305.716,Z 414.747,A -85,B 0,C 180,E1 -16145.08,E2 -16145.08} C_VEL
LIN {X 0,Y 305.964,Z 411.208,A -85,B 0,C 180,E1 -16148.649,E2 -16148.649} C_VEL
LIN {X 0,Y 305.878,Z 408.29,A -85,B 0,C 180,E1 -16151.784,E2 -16151.784} C_VEL
LIN {X 0,Y 305.443,Z 405.068,A -85,B 0,C 180,E1 -16155.503,E2 -16155.503} C_VEL
LIN {X 0,Y 305.457,Z 405.064,A -85,B 0,C 180,E1 -16159.4,E2 -16159.4} C_VEL
LIN {X 0,Y 305.477,Z 405.059,A -85,B 0,C 180,E1 -16163.261,E2 -16163.261} C_VEL
LIN {X 0,Y 305.467,Z 405.061,A -85,B 0,C 180,E1 -16166.483,E2 -16166.483} C_VEL
LIN {X 0,Y 305.466,Z 405.06,A -85,B 0,C 180,E1 -16169.591,E2 -16169.591} C_VEL
LIN {X 0,Y 305.523,Z 405.054,A -85,B 0,C 180,E1 -16172.609,E2 -16172.609} C_VEL
LIN {X 0,Y 305.51,Z 405.054,A -85,B 0,C 180,E1 -16175.539,E2 -16175.539} C_VEL
LIN {X 0,Y 305.523,Z 405.047,A -85,B 0,C 180,E1 -16179.815,E2 -16179.815} C_VEL
LIN {X 0,Y 305.577,Z 405.047,A -85,B 0,C 180,E1 -16182.603,E2 -16182.603} C_VEL
LIN {X 0,Y 305.604,Z 405.041,A -85,B 0,C 180,E1 -16184.384,E2 -16184.384} C_VEL
LIN {X 0,Y 304.959,Z 405.125,A -85,B 0,C 180,E1 -16185.484,E2 -16185.484} C_VEL
LIN {X 0,Y 302.089,Z 405.483,A -85,B 0,C 180,E1 -16187.274,E2 -16187.274} C_VEL
LIN {X 0,Y 299.677,Z 405.781,A -85,B 0,C 180,E1 -16188.726,E2 -16188.726} C_VEL
LIN {X 0,Y 298.699,Z 405.903,A -85,B 0,C 180,E1 -16189.852,E2 -16189.852} C_VEL
LIN {X 0,Y 298.651,Z 405.907,A -85,B 0,C 180,E1 -16190.233,E2 -16190.233} C_VEL
LIN {X 0,Y 298.801,Z 405.891,A -85,B 0,C 180,E1 -16193.246,E2 -16193.246} C_VEL
LIN {X 0,Y 298.925,Z 405.875,A -85,B 0,C 180,E1 -16198.653,E2 -16198.653} C_VEL
LIN {X 0,Y 298.927,Z 405.873,A -85,B 0,C 180,E1 -16201.347,E2 -16201.347} C_VEL
LIN {X 0,Y 298.801,Z 405.892,A -85,B 0,C 180,E1 -16206.754,E2 -16206.754} C_VEL
LIN {X 0,Y 298.683,Z 405.906,A -85,B 0,C 180,E1 -16209.48,E2 -16209.48} C_VEL
LIN {X 0,Y 298.555,Z 405.921,A -85,B 0,C 180,E1 -16213.615,E2 -16213.615} C_VEL
LIN {X 0,Y 298.551,Z 405.922,A -85,B 0,C 180,E1 -16216.408,E2 -16216.408} C_VEL
LIN {X 0,Y 298.515,Z 405.927,A -85,B 0,C 180,E1 -16219.655,E2 -16219.655} C_VEL
LIN {X 0,Y 298.459,Z 405.928,A -85,B 0,C 180,E1 -16223.597,E2 -16223.597} C_VEL
LIN {X 0,Y 298.488,Z 405.927,A -85,B 0,C 180,E1 -16226.574,E2 -16226.574} C_VEL
LIN {X 0,Y 298.418,Z 405.935,A -85,B 0,C 180,E1 -16229.641,E2 -16229.641} C_VEL
LIN {X 0,Y 298.397,Z 405.942,A -85,B 0,C 180,E1 -16232.8,E2 -16232.8} C_VEL
LIN {X 0,Y 298.472,Z 405.936,A -85,B 0,C 180,E1 -16236.814,E2 -16236.814} C_VEL
LIN {X 0,Y 298.432,Z 405.963,A -85,B 0,C 180,E1 -16241.097,E2 -16241.097} C_VEL
LIN {X 0,Y 298.963,Z 409.308,A -85,B 0,C 180,E1 -16244.849,E2 -16244.849} C_VEL
LIN {X 0,Y 299.26,Z 411.403,A -85,B 0,C 180,E1 -16247.074,E2 -16247.074} C_VEL
LIN {X 0,Y 299.414,Z 413.218,A -85,B 0,C 180,E1 -16248.911,E2 -16248.911} C_VEL
LIN {X 0,Y 299.466,Z 415.128,A -85,B 0,C 180,E1 -16250.756,E2 -16250.756} C_VEL
LIN {X 0,Y 299.13,Z 418.683,A -85,B 0,C 180,E1 -16254.029,E2 -16254.029} C_VEL
LIN {X 0,Y 298.642,Z 422.318,A -85,B 0,C 180,E1 -16257.23,E2 -16257.23} C_VEL
LIN {X 0,Y 298.315,Z 425.677,A -85,B 0,C 180,E1 -16259.994,E2 -16259.994} C_VEL
LIN {X 0,Y 299.233,Z 428.72,A -85,B 0,C 180,E1 -16260.193,E2 -16260.193} C_VEL
LIN {X 0,Y 303.434,Z 441.512,A -85,B 0,C 180,E1 -16261.2,E2 -16261.2} C_VEL
LIN {X 0,Y 306.916,Z 455.25,A -85,B 0,C 180,E1 -16262.415,E2 -16262.415} C_VEL
LIN {X 0,Y 309.178,Z 467.597,A -85,B 0,C 180,E1 -16263.655,E2 -16263.655} C_VEL
LIN {X 0,Y 310.277,Z 478.052,A -85,B 0,C 180,E1 -16264.821,E2 -16264.821} C_VEL
LIN {X 0,Y 308.403,Z 489.956,A -85,B 0,C 180,E1 -16266.14,E2 -16266.14} C_VEL
LIN {X 0,Y 306.164,Z 501.704,A -85,B 0,C 180,E1 -16267.743,E2 -16267.743} C_VEL
LIN {X 0,Y 304.267,Z 511.433,A -85,B 0,C 180,E1 -16269.375,E2 -16269.375} C_VEL
LIN {X 0,Y 302.266,Z 521.166,A -85,B 0,C 180,E1 -16271.355,E2 -16271.355} C_VEL
LIN {X 0,Y 300.466,Z 529.902,A -85,B 0,C 180,E1 -16273.537,E2 -16273.537} C_VEL
LIN {X 0,Y 299.224,Z 536.982,A -85,B 0,C 180,E1 -16275.722,E2 -16275.722} C_VEL
LIN {X 0,Y 298.07,Z 542.382,A -85,B 0,C 180,E1 -16277.748,E2 -16277.748} C_VEL
LIN {X 0,Y 297.216,Z 548.067,A -85,B 0,C 180,E1 -16280.472,E2 -16280.472} C_VEL
LIN {X 0,Y 296.69,Z 552.191,A -85,B 0,C 180,E1 -16283.198,E2 -16283.198} C_VEL
LIN {X 0,Y 296.486,Z 554.884,A -85,B 0,C 180,E1 -16285.922,E2 -16285.922} C_VEL
LIN {X 0,Y 296.447,Z 556.216,A -85,B 0,C 180,E1 -16288.641,E2 -16288.641} C_VEL
LIN {X 0,Y 296.447,Z 556.211,A -85,B 0,C 180,E1 -16291.358,E2 -16291.358} C_VEL
LIN {X 0,Y 296.487,Z 554.871,A -85,B 0,C 180,E1 -16294.078,E2 -16294.078} C_VEL
LIN {X 0,Y 296.694,Z 552.169,A -85,B 0,C 180,E1 -16296.802,E2 -16296.802} C_VEL
LIN {X 0,Y 297.2,Z 548.03,A -85,B 0,C 180,E1 -16299.528,E2 -16299.528} C_VEL
LIN {X 0,Y 298.068,Z 542.332,A -85,B 0,C 180,E1 -16302.252,E2 -16302.252} C_VEL
LIN {X 0,Y 299.397,Z 535.91,A -85,B 0,C 180,E1 -16304.616,E2 -16304.616} C_VEL
LIN {X 0,Y 300.895,Z 527.934,A -85,B 0,C 180,E1 -16306.975,E2 -16306.975} C_VEL
LIN {X 0,Y 302.564,Z 519.585,A -85,B 0,C 180,E1 -16308.977,E2 -16308.977} C_VEL
LIN {X 0,Y 304.657,Z 509.537,A -85,B 0,C 180,E1 -16310.951,E2 -16310.951} C_VEL
LIN {X 0,Y 306.859,Z 498.324,A -85,B 0,C 180,E1 -16312.736,E2 -16312.736} C_VEL
LIN {X 0,Y 309.001,Z 485.994,A -85,B 0,C 180,E1 -16314.314,E2 -16314.314} C_VEL
LIN {X 0,Y 310.218,Z 476.351,A -85,B 0,C 180,E1 -16315.353,E2 -16315.353} C_VEL
LIN {X 0,Y 308.551,Z 463.613,A -85,B 0,C 180,E1 -16316.741,E2 -16316.741} C_VEL
LIN {X 0,Y 305.71,Z 450.194,A -85,B 0,C 180,E1 -16318.033,E2 -16318.033} C_VEL
LIN {X 0,Y 301.718,Z 435.894,A -85,B 0,C 180,E1 -16319.228,E2 -16319.228} C_VEL
LIN {X 0,Y 298.346,Z 426.069,A -85,B 0,C 180,E1 -16319.961,E2 -16319.961} C_VEL
LIN {X 0,Y 298.293,Z 425.472,A -85,B 0,C 180,E1 -16320.041,E2 -16320.041} C_VEL
LIN {X 0,Y 298.952,Z 420.146,A -85,B 0,C 180,E1 -16324.633,E2 -16324.633} C_VEL
LIN {X 0,Y 299.315,Z 416.815,A -85,B 0,C 180,E1 -16327.625,E2 -16327.625} C_VEL
LIN {X 0,Y 299.457,Z 415.013,A -85,B 0,C 180,E1 -16329.321,E2 -16329.321} C_VEL
LIN {X 0,Y 299.402,Z 412.971,A -85,B 0,C 180,E1 -16331.31,E2 -16331.31} C_VEL
LIN {X 0,Y 299.003,Z 409.556,A -85,B 0,C 180,E1 -16334.841,E2 -16334.841} C_VEL
LIN {X 0,Y 298.727,Z 407.602,A -85,B 0,C 180,E1 -16336.979,E2 -16336.979} C_VEL
LIN {X 0,Y 298.43,Z 405.94,A -85,B 0,C 180,E1 -16338.903,E2 -16338.903} C_VEL
LIN {X 0,Y 298.471,Z 405.933,A -85,B 0,C 180,E1 -16343.186,E2 -16343.186} C_VEL
LIN {X 0,Y 298.396,Z 405.943,A -85,B 0,C 180,E1 -16347.2,E2 -16347.2} C_VEL
LIN {X 0,Y 298.428,Z 405.939,A -85,B 0,C 180,E1 -16350.616,E2 -16350.616} C_VEL
LIN {X 0,Y 298.483,Z 405.931,A -85,B 0,C 180,E1 -16353.475,E2 -16353.475} C_VEL
LIN {X 0,Y 298.431,Z 405.936,A -85,B 0,C 180,E1 -16356.699,E2 -16356.699} C_VEL
LIN {X 0,Y 298.539,Z 405.924,A -85,B 0,C 180,E1 -16360.757,E2 -16360.757} C_VEL
LIN {X 0,Y 298.595,Z 405.914,A -85,B 0,C 180,E1 -16364.995,E2 -16364.995} C_VEL
LIN {X 0,Y 298.595,Z 405.912,A -85,B 0,C 180,E1 -16369.147,E2 -16369.147} C_VEL
LIN {X 0,Y 298.76,Z 405.893,A -85,B 0,C 180,E1 -16371.886,E2 -16371.886} C_VEL
LIN {X 0,Y 298.662,Z 405.907,A -85,B 0,C 180,E1 -16374.599,E2 -16374.599} C_VEL
LIN {X 0,Y 298.925,Z 405.876,A -85,B 0,C 180,E1 -16378.653,E2 -16378.653} C_VEL
LIN {X 0,Y 298.925,Z 405.876,A -85,B 0,C 180,E1 -16381.347,E2 -16381.347} C_VEL
LIN {X 0,Y 298.799,Z 405.891,A -85,B 0,C 180,E1 -16386.754,E2 -16386.754} C_VEL
LIN {X 0,Y 298.682,Z 405.906,A -85,B 0,C 180,E1 -16389.481,E2 -16389.481} C_VEL
LIN {X 0,Y 298.554,Z 405.916,A -85,B 0,C 180,E1 -16393.615,E2 -16393.615} C_VEL
LIN {X 0,Y 298.55,Z 405.919,A -85,B 0,C 180,E1 -16396.409,E2 -16396.409} C_VEL
LIN {X 0,Y 298.514,Z 405.927,A -85,B 0,C 180,E1 -16399.655,E2 -16399.655} C_VEL
LIN {X 0,Y 298.459,Z 405.933,A -85,B 0,C 180,E1 -16403.598,E2 -16403.598} C_VEL
LIN {X 0,Y 298.49,Z 405.929,A -85,B 0,C 180,E1 -16406.574,E2 -16406.574} C_VEL
LIN {X 0,Y 298.418,Z 405.938,A -85,B 0,C 180,E1 -16409.642,E2 -16409.642} C_VEL
LIN {X 0,Y 298.396,Z 405.942,A -85,B 0,C 180,E1 -16412.8,E2 -16412.8} C_VEL
LIN {X 0,Y 298.466,Z 405.933,A -85,B 0,C 180,E1 -16416.813,E2 -16416.813} C_VEL
LIN {X 0,Y 298.388,Z 405.942,A -85,B 0,C 180,E1 -16421.088,E2 -16421.088} C_VEL
LIN {X 0,Y 298.399,Z 405.942,A -85,B 0,C 180,E1 -16423.103,E2 -16423.103} C_VEL
LIN {X 0,Y 298.482,Z 406.627,A -85,B 0,C 180,E1 -16425.059,E2 -16425.059} C_VEL
LIN {X 0,Y 298.902,Z 409.867,A -85,B 0,C 180,E1 -16428.825,E2 -16428.825} C_VEL
LIN {X 0,Y 298.87,Z 413.09,A -85,B 0,C 180,E1 -16432.31,E2 -16432.31} C_VEL
LIN {X 0,Y 298.64,Z 416.3,A -85,B 0,C 180,E1 -16435.612,E2 -16435.612} C_VEL
LIN {X 0,Y 298.179,Z 420.354,A -85,B 0,C 180,E1 -16439.553,E2 -16439.553} C_VEL
LIN {X 0,Y 298.127,Z 420.855,A -85,B 0,C 180,E1 -16440.035,E2 -16440.035} C_VEL
LIN {X 0,Y 299.22,Z 424.214,A -85,B 0,C 180,E1 -16440.283,E2 -16440.283} C_VEL
LIN {X 0,Y 303.931,Z 437.802,A -85,B 0,C 180,E1 -16441.4,E2 -16441.4} C_VEL
LIN {X 0,Y 307.202,Z 449.986,A -85,B 0,C 180,E1 -16442.516,E2 -16442.516} C_VEL
LIN {X 0,Y 309.796,Z 462.803,A -85,B 0,C 180,E1 -16443.835,E2 -16443.835} C_VEL
LIN {X 0,Y 310.783,Z 470.633,A -85,B 0,C 180,E1 -16444.711,E2 -16444.711} C_VEL
LIN {X 0,Y 309.019,Z 482.701,A -85,B 0,C 180,E1 -16446.013,E2 -16446.013} C_VEL
LIN {X 0,Y 306.813,Z 494.725,A -85,B 0,C 180,E1 -16447.616,E2 -16447.616} C_VEL
LIN {X 0,Y 305.005,Z 503.787,A -85,B 0,C 180,E1 -16449.075,E2 -16449.075} C_VEL
LIN {X 0,Y 302.95,Z 513.84,A -85,B 0,C 180,E1 -16451.048,E2 -16451.048} C_VEL
LIN {X 0,Y 301.114,Z 522.497,A -85,B 0,C 180,E1 -16453.126,E2 -16453.126} C_VEL
LIN {X 0,Y 299.738,Z 530.156,A -85,B 0,C 180,E1 -16455.401,E2 -16455.401} C_VEL
LIN {X 0,Y 298.35,Z 536.573,A -85,B 0,C 180,E1 -16457.76,E2 -16457.76} C_VEL
LIN {X 0,Y 297.39,Z 542.261,A -85,B 0,C 180,E1 -16460.478,E2 -16460.478} C_VEL
LIN {X 0,Y 296.854,Z 546.393,A -85,B 0,C 180,E1 -16463.202,E2 -16463.202} C_VEL
LIN {X 0,Y 296.574,Z 549.095,A -85,B 0,C 180,E1 -16465.923,E2 -16465.923} C_VEL
LIN {X 0,Y 296.46,Z 550.447,A -85,B 0,C 180,E1 -16468.642,E2 -16468.642} C_VEL
LIN {X 0,Y 296.459,Z 550.477,A -85,B 0,C 180,E1 -16471.359,E2 -16471.359} C_VEL
LIN {X 0,Y 296.573,Z 549.182,A -85,B 0,C 180,E1 -16474.077,E2 -16474.077} C_VEL
LIN {X 0,Y 296.854,Z 546.532,A -85,B 0,C 180,E1 -16476.798,E2 -16476.798} C_VEL
LIN {X 0,Y 297.376,Z 542.46,A -85,B 0,C 180,E1 -16479.523,E2 -16479.523} C_VEL
LIN {X 0,Y 298.323,Z 536.833,A -85,B 0,C 180,E1 -16482.241,E2 -16482.241} C_VEL
LIN {X 0,Y 299.706,Z 530.478,A -85,B 0,C 180,E1 -16484.601,E2 -16484.601} C_VEL
LIN {X 0,Y 301.119,Z 522.878,A -85,B 0,C 180,E1 -16486.878,E2 -16486.878} C_VEL
LIN {X 0,Y 302.896,Z 514.314,A -85,B 0,C 180,E1 -16488.956,E2 -16488.956} C_VEL
LIN {X 0,Y 304.942,Z 504.354,A -85,B 0,C 180,E1 -16490.93,E2 -16490.93} C_VEL
LIN {X 0,Y 307.177,Z 493.263,A -85,B 0,C 180,E1 -16492.712,E2 -16492.712} C_VEL
LIN {X 0,Y 309.131,Z 482.221,A -85,B 0,C 180,E1 -16494.156,E2 -16494.156} C_VEL
LIN {X 0,Y 310.857,Z 470.231,A -85,B 0,C 180,E1 -16495.44,E2 -16495.44} C_VEL
LIN {X 0,Y 308.747,Z 457.113,A -85,B 0,C 180,E1 -16496.89,E2 -16496.89} C_VEL
LIN {X 0,Y 305.597,Z 443.727,A -85,B 0,C 180,E1 -16498.192,E2 -16498.192} C_VEL
LIN {X 0,Y 301.7,Z 430.876,A -85,B 0,C 180,E1 -16499.299,E2 -16499.299} C_VEL
LIN {X 0,Y 298.272,Z 421.888,A -85,B 0,C 180,E1 -16500.016,E2 -16500.016} C_VEL
LIN {X 0,Y 298.092,Z 420.833,A -85,B 0,C 180,E1 -16500.097,E2 -16500.097} C_VEL
LIN {X 0,Y 298.42,Z 418.042,A -85,B 0,C 180,E1 -16502.797,E2 -16502.797} C_VEL
LIN {X 0,Y 298.782,Z 414.806,A -85,B 0,C 180,E1 -16506.019,E2 -16506.019} C_VEL
LIN {X 0,Y 298.944,Z 411.583,A -85,B 0,C 180,E1 -16509.402,E2 -16509.402} C_VEL
LIN {X 0,Y 298.921,Z 409.934,A -85,B 0,C 180,E1 -16511.205,E2 -16511.205} C_VEL
LIN {X 0,Y 298.516,Z 406.634,A -85,B 0,C 180,E1 -16515.066,E2 -16515.066} C_VEL
LIN {X 0,Y 298.405,Z 405.946,A -85,B 0,C 180,E1 -16516.921,E2 -16516.921} C_VEL
LIN {X 0,Y 298.406,Z 405.941,A -85,B 0,C 180,E1 -16521.006,E2 -16521.006} C_VEL
LIN {X 0,Y 298.421,Z 405.937,A -85,B 0,C 180,E1 -16523.93,E2 -16523.93} C_VEL
LIN {X 0,Y 298.398,Z 405.939,A -85,B 0,C 180,E1 -16527.983,E2 -16527.983} C_VEL
LIN {X 0,Y 298.466,Z 405.932,A -85,B 0,C 180,E1 -16531.904,E2 -16531.904} C_VEL
LIN {X 0,Y 298.488,Z 405.929,A -85,B 0,C 180,E1 -16534.924,E2 -16534.924} C_VEL
LIN {X 0,Y 298.454,Z 405.928,A -85,B 0,C 180,E1 -16539.315,E2 -16539.315} C_VEL
LIN {X 0,Y 298.541,Z 405.923,A -85,B 0,C 180,E1 -16542.179,E2 -16542.179} C_VEL
LIN {X 0,Y 298.596,Z 405.915,A -85,B 0,C 180,E1 -16544.995,E2 -16544.995} C_VEL
LIN {X 0,Y 298.597,Z 405.916,A -85,B 0,C 180,E1 -16549.147,E2 -16549.147} C_VEL
LIN {X 0,Y 298.651,Z 405.907,A -85,B 0,C 180,E1 -16550.233,E2 -16550.233} C_VEL
LIN {X 0,Y 298.384,Z 405.943,A -85,B 0,C 180,E1 -16550.986,E2 -16550.986} C_VEL
LIN {X 0,Y 297.031,Z 406.113,A -85,B 0,C 180,E1 -16552.097,E2 -16552.097} C_VEL
LIN {X 0,Y 292.623,Z 406.66,A -85,B 0,C 180,E1 -16554.678,E2 -16554.678} C_VEL
LIN {X 0,Y 291.637,Z 406.78,A -85,B 0,C 180,E1 -16555.832,E2 -16555.832} C_VEL
LIN {X 0,Y 291.601,Z 406.783,A -85,B 0,C 180,E1 -16556.223,E2 -16556.223} C_VEL
LIN {X 0,Y 291.891,Z 406.751,A -85,B 0,C 180,E1 -16558.62,E2 -16558.62} C_VEL
LIN {X 0,Y 291.893,Z 406.75,A -85,B 0,C 180,E1 -16561.38,E2 -16561.38} C_VEL
LIN {X 0,Y 291.749,Z 406.769,A -85,B 0,C 180,E1 -16566.918,E2 -16566.918} C_VEL
LIN {X 0,Y 291.632,Z 406.784,A -85,B 0,C 180,E1 -16569.712,E2 -16569.712} C_VEL
LIN {X 0,Y 291.525,Z 406.797,A -85,B 0,C 180,E1 -16573.95,E2 -16573.95} C_VEL
LIN {X 0,Y 291.489,Z 406.799,A -85,B 0,C 180,E1 -16576.818,E2 -16576.818} C_VEL
LIN {X 0,Y 291.453,Z 406.807,A -85,B 0,C 180,E1 -16579.875,E2 -16579.875} C_VEL
LIN {X 0,Y 291.402,Z 406.806,A -85,B 0,C 180,E1 -16584.205,E2 -16584.205} C_VEL
LIN {X 0,Y 291.422,Z 406.805,A -85,B 0,C 180,E1 -16587.272,E2 -16587.272} C_VEL
LIN {X 0,Y 291.336,Z 406.817,A -85,B 0,C 180,E1 -16590.437,E2 -16590.437} C_VEL
LIN {X 0,Y 291.347,Z 406.822,A -85,B 0,C 180,E1 -16593.698,E2 -16593.698} C_VEL
LIN {X 0,Y 291.406,Z 406.816,A -85,B 0,C 180,E1 -16597.261,E2 -16597.261} C_VEL
LIN {X 0,Y 291.387,Z 406.874,A -85,B 0,C 180,E1 -16600.633,E2 -16600.633} C_VEL
LIN {X 0,Y 291.874,Z 410.016,A -85,B 0,C 180,E1 -16604.29,E2 -16604.29} C_VEL
LIN {X 0,Y 292.293,Z 413.161,A -85,B 0,C 180,E1 -16607.682,E2 -16607.682} C_VEL
LIN {X 0,Y 292.428,Z 415.706,A -85,B 0,C 180,E1 -16610.27,E2 -16610.27} C_VEL
LIN {X 0,Y 292.226,Z 418.614,A -85,B 0,C 180,E1 -16613.04,E2 -16613.04} C_VEL
LIN {X 0,Y 291.736,Z 422.251,A -85,B 0,C 180,E1 -16616.353,E2 -16616.353} C_VEL
LIN {X 0,Y 291.322,Z 425.451,A -85,B 0,C 180,E1 -16619.173,E2 -16619.173} C_VEL
LIN {X 0,Y 292.449,Z 428.966,A -85,B 0,C 180,E1 -16619.439,E2 -16619.439} C_VEL
LIN {X 0,Y 296.858,Z 442.369,A -85,B 0,C 180,E1 -16620.549,E2 -16620.549} C_VEL
